// cont log-messages
      L     "SSA_LOG_Value_Queue".Input.Para_0099;	// message counter
      L     1;
      +I;
      T     "SSA_LOG_Value_Queue".Input.Para_0099;	// message counter
// Transform Basic Time to Local Time 
//      CALL  "BT_LT"
//       BT     :="DB Prozesszeit".Arbeitsbereich.dt1
//       WS_DAT :="RegelDB"
//       RET_VAL:=MW218
//       LT     :="RegelDB".LocalTime
// put timestamp into message
      CALL  FC 49 (
           $1                       := 1010,
           $2                       := 18,
           $3                       := 1005,
           $4                       := 462,
           $5                       := 8,
           $6                       := P#M 210.0);
///
      CALL  "SSA_MH_LogEntry_ActValue" (
           DBNumber                 := 1005);
E060: NOP   0;
///     
// Ereignis 26  Kommt         
      A     #EREIGNISBIT_26;
      FP    #Ereignis_26.FP_Kommt;
      JCN   E061;
// header
      L     #MessageType;
      T     "SSA_LOG_Value_Queue".Input.Header.SecType;	// type
      L     #MessageFormat;
      T     "SSA_LOG_Value_Queue".Input.Header.Format;	// format
      L     #JobNumber;
      T     "SSA_LOG_Value_Queue".Input.Para_0005;
      L     #processMinute;
      T     "SSA_LOG_Value_Queue".Input.Para_0007;
      L     #StepNumber;
      T     "SSA_LOG_Value_Queue".Input.Para_0008;
      L     #StepTimeMin;
      T     "SSA_LOG_Value_Queue".Input.Para_0009;
// values integer
      L     #EventObject_26;	// event-Nr
      T     "SSA_LOG_Value_Queue".Input.Para_0010;
      L     1;	// object-state coming
      T     "SSA_LOG_Value_Queue".Input.Para_0011;
      L     0;	// number additional param
      T     "SSA_LOG_Value_Queue".Input.Para_0012;
// cont log-messages
      L     "SSA_LOG_Value_Queue".Input.Para_0099;	// message counter
      L     1;
      +I;
      T     "SSA_LOG_Value_Queue".Input.Para_0099;	// message counter
// Transform Basic Time to Local Time 
//      CALL  "BT_LT"
//       BT     :="DB Prozesszeit".Arbeitsbereich.dt1
//       WS_DAT :="RegelDB"
//       RET_VAL:=MW218
//       LT     :="RegelDB".LocalTime
// put timestamp into message
      CALL  FC 49 (
           $1                       := 1010,
           $2                       := 18,
           $3                       := 1005,
           $4                       := 462,
           $5                       := 8,
           $6                       := P#M 210.0);
///
      CALL  "SSA_MH_LogEntry_ActValue" (
           DBNumber                 := 1005);
E061: NOP   0;
///
// Ereignis 26  Geht        
      A     #EREIGNISBIT_26;
      FN    #Ereignis_26.FN_Geht;
      JCN   E062;
// header
      L     #MessageType;
      T     "SSA_LOG_Value_Queue".Input.Header.SecType;	// type
      L     #MessageFormat;
      T     "SSA_LOG_Value_Queue".Input.Header.Format;	// format
      L     #JobNumber;
      T     "SSA_LOG_Value_Queue".Input.Para_0005;
      L     #processMinute;
      T     "SSA_LOG_Value_Queue".Input.Para_0007;
      L     #StepNumber;
      T     "SSA_LOG_Value_Queue".Input.Para_0008;
      L     #StepTimeMin;
      T     "SSA_LOG_Value_Queue".Input.Para_0009;
// values integer
      L     #EventObject_26;	// event-Nr
      T     "SSA_LOG_Value_Queue".Input.Para_0010;
      L     2;	// object-state going
      T     "SSA_LOG_Value_Queue".Input.Para_0011;
      L     0;	// number additional param
      T     "SSA_LOG_Value_Queue".Input.Para_0012;
// cont log-messages
      L     "SSA_LOG_Value_Queue".Input.Para_0099;	// message counter
      L     1;
      +I;
      T     "SSA_LOG_Value_Queue".Input.Para_0099;	// message counter
// Transform Basic Time to Local Time 
//      CALL  "BT_LT"
//       BT     :="DB Prozesszeit".Arbeitsbereich.dt1
//       WS_DAT :="RegelDB"
//       RET_VAL:=MW218
//       LT     :="RegelDB".LocalTime
// put timestamp into message
      CALL  FC 49 (
           $1                       := 1010,
           $2                       := 18,
           $3                       := 1005,
           $4                       := 462,
           $5                       := 8,
           $6                       := P#M 210.0);
///
      CALL  "SSA_MH_LogEntry_ActValue" (
           DBNumber                 := 1005);
E062: NOP   0;
///     
// Ereignis 27  Kommt         
      A     #EREIGNISBIT_27;
      FP    #Ereignis_27.FP_Kommt;
      JCN   E063;
/// header
      L     #MessageType;
      T     "SSA_LOG_Value_Queue".Input.Header.SecType;	// type
      L     #MessageFormat;
      T     "SSA_LOG_Value_Queue".Input.Header.Format;	// format
      L     #JobNumber;
      T     "SSA_LOG_Value_Queue".Input.Para_0005;
      L     #processMinute;
      T     "SSA_LOG_Value_Queue".Input.Para_0007;
      L     #StepNumber;
      T     "SSA_LOG_Value_Queue".Input.Para_0008;
      L     #StepTimeMin;
      T     "SSA_LOG_Value_Queue".Input.Para_0009;
// values integer
      L     #EventObject_27;	// event-Nr
      T     "SSA_LOG_Value_Queue".Input.Para_0010;
      L     1;	// object-state coming
      T     "SSA_LOG_Value_Queue".Input.Para_0011;
      L     0;	// number additional param
      T     "SSA_LOG_Value_Queue".Input.Para_0012;
// cont log-messages
      L     "SSA_LOG_Value_Queue".Input.Para_0099;	// message counter
      L     1;
      +I;
      T     "SSA_LOG_Value_Queue".Input.Para_0099;	// message counter
// Transform Basic Time to Local Time 
//      CALL  "BT_LT"
//       BT     :="DB Prozesszeit".Arbeitsbereich.dt1
//       WS_DAT :="RegelDB"
//       RET_VAL:=MW218
//       LT     :="RegelDB".LocalTime
// put timestamp into message
      CALL  FC 49 (
           $1                       := 1010,
           $2                       := 18,
           $3                       := 1005,
           $4                       := 462,
           $5                       := 8,
           $6                       := P#M 210.0);
///
      CALL  "SSA_MH_LogEntry_ActValue" (
           DBNumber                 := 1005);
E063: NOP   0;
///
// Ereignis 27  Geht        
      A     #EREIGNISBIT_27;
      FN    #Ereignis_27.FN_Geht;
      JCN   E064;
// header
      L     #MessageType;
      T     "SSA_LOG_Value_Queue".Input.Header.SecType;	// type
      L     #MessageFormat;
      T     "SSA_LOG_Value_Queue".Input.Header.Format;	// format
      L     #JobNumber;
      T     "SSA_LOG_Value_Queue".Input.Para_0005;
      L     #processMinute;
      T     "SSA_LOG_Value_Queue".Input.Para_0007;
      L     #StepNumber;
      T     "SSA_LOG_Value_Queue".Input.Para_0008;
      L     #StepTimeMin;
      T     "SSA_LOG_Value_Queue".Input.Para_0009;
// values integer
      L     #EventObject_27;	// event-Nr
      T     "SSA_LOG_Value_Queue".Input.Para_0010;
      L     2;	// object-state going
      T     "SSA_LOG_Value_Queue".Input.Para_0011;
      L     0;	// number additional param
      T     "SSA_LOG_Value_Queue".Input.Para_0012;
// cont log-messages
      L     "SSA_LOG_Value_Queue".Input.Para_0099;	// message counter
      L     1;
      +I;
      T     "SSA_LOG_Value_Queue".Input.Para_0099;	// message counter
// Transform Basic Time to Local Time 
//      CALL  "BT_LT"
//       BT     :="DB Prozesszeit".Arbeitsbereich.dt1
//       WS_DAT :="RegelDB"
//       RET_VAL:=MW218
//       LT     :="RegelDB".LocalTime
// put timestamp into message
      CALL  FC 49 (
           $1                       := 1010,
           $2                       := 18,
           $3                       := 1005,
           $4                       := 462,
           $5                       := 8,
           $6                       := P#M 210.0);
///
      CALL  "SSA_MH_LogEntry_ActValue" (
           DBNumber                 := 1005);
E064: NOP   0;
///     
// Ereignis 28  Kommt         
      A     #EREIGNISBIT_28;
      FP    #Ereignis_28.FP_Kommt;
      JCN   E065;
// header
      L     #MessageType;
      T     "SSA_LOG_Value_Queue".Input.Header.SecType;	// type
      L     #MessageFormat;
      T     "SSA_LOG_Value_Queue".Input.Header.Format;	// format
      L     #JobNumber;
      T     "SSA_LOG_Value_Queue".Input.Para_0005;
      L     #processMinute;
      T     "SSA_LOG_Value_Queue".Input.Para_0007;
      L     #StepNumber;
      T     "SSA_LOG_Value_Queue".Input.Para_0008;
      L     #StepTimeMin;
      T     "SSA_LOG_Value_Queue".Input.Para_0009;
// values integer
      L     #EventObject_28;	// event-Nr
      T     "SSA_LOG_Value_Queue".Input.Para_0010;
      L     1;	// object-state coming
      T     "SSA_LOG_Value_Queue".Input.Para_0011;
      L     0;	// number additional param
      T     "SSA_LOG_Value_Queue".Input.Para_0012;
// cont log-messages
      L     "SSA_LOG_Value_Queue".Input.Para_0099;	// message counter
      L     1;
      +I;
      T     "SSA_LOG_Value_Queue".Input.Para_0099;	// message counter
// Transform Basic Time to Local Time 
//      CALL  "BT_LT"
//       BT     :="DB Prozesszeit".Arbeitsbereich.dt1
//       WS_DAT :="RegelDB"
//       RET_VAL:=MW218
//       LT     :="RegelDB".LocalTime
// put timestamp into message
      CALL  FC 49 (
           $1                       := 1010,
           $2                       := 18,
           $3                       := 1005,
           $4                       := 462,
           $5                       := 8,
           $6                       := P#M 210.0);
///
      CALL  "SSA_MH_LogEntry_ActValue" (
           DBNumber                 := 1005);
E065: NOP   0;
///
// Ereignis 28  Geht        
      A     #EREIGNISBIT_28;
      FN    #Ereignis_28.FN_Geht;
      JCN   E066;
// header
      L     #MessageType;
      T     "SSA_LOG_Value_Queue".Input.Header.SecType;	// type
      L     #MessageFormat;
      T     "SSA_LOG_Value_Queue".Input.Header.Format;	// format
      L     #JobNumber;
      T     "SSA_LOG_Value_Queue".Input.Para_0005;
      L     #processMinute;
      T     "SSA_LOG_Value_Queue".Input.Para_0007;
      L     #StepNumber;
      T     "SSA_LOG_Value_Queue".Input.Para_0008;
      L     #StepTimeMin;
      T     "SSA_LOG_Value_Queue".Input.Para_0009;
// values integer
      L     #EventObject_28;	// event-Nr
      T     "SSA_LOG_Value_Queue".Input.Para_0010;
      L     2;	// object-state going
      T     "SSA_LOG_Value_Queue".Input.Para_0011;
      L     0;	// number additional param
      T     "SSA_LOG_Value_Queue".Input.Para_0012;
// cont log-messages
      L     "SSA_LOG_Value_Queue".Input.Para_0099;	// message counter
      L     1;
      +I;
      T     "SSA_LOG_Value_Queue".Input.Para_0099;	// message counter
// Transform Basic Time to Local Time 
//      CALL  "BT_LT"
//       BT     :="DB Prozesszeit".Arbeitsbereich.dt1
//       WS_DAT :="RegelDB"
//       RET_VAL:=MW218
//       LT     :="RegelDB".LocalTime
// put timestamp into message
      CALL  FC 49 (
           $1                       := 1010,
           $2                       := 18,
           $3                       := 1005,
           $4                       := 462,
           $5                       := 8,
           $6                       := P#M 210.0);
///
      CALL  "SSA_MH_LogEntry_ActValue" (
           DBNumber                 := 1005);
E066: NOP   0;
///     
// Ereignis 29  Kommt         
      A     #EREIGNISBIT_29;
      FP    #Ereignis_29.FP_Kommt;
      JCN   E067;
// header
      L     #MessageType;
      T     "SSA_LOG_Value_Queue".Input.Header.SecType;	// type
      L     #MessageFormat;
      T     "SSA_LOG_Value_Queue".Input.Header.Format;	// format
      L     #JobNumber;
      T     "SSA_LOG_Value_Queue".Input.Para_0005;
      L     #processMinute;
      T     "SSA_LOG_Value_Queue".Input.Para_0007;
      L     #StepNumber;
      T     "SSA_LOG_Value_Queue".Input.Para_0008;
      L     #StepTimeMin;
      T     "SSA_LOG_Value_Queue".Input.Para_0009;
// values integer
      L     #EventObject_29;	// event-Nr
      T     "SSA_LOG_Value_Queue".Input.Para_0010;
      L     1;	// object-state coming
      T     "SSA_LOG_Value_Queue".Input.Para_0011;
      L     0;	// number additional param
      T     "SSA_LOG_Value_Queue".Input.Para_0012;
// cont log-messages
      L     "SSA_LOG_Value_Queue".Input.Para_0099;	// message counter
      L     1;
      +I;
      T     "SSA_LOG_Value_Queue".Input.Para_0099;	// message counter
// Transform Basic Time to Local Time 
//      CALL  "BT_LT"
//       BT     :="DB Prozesszeit".Arbeitsbereich.dt1
//       WS_DAT :="RegelDB"
//       RET_VAL:=MW218
//       LT     :="RegelDB".LocalTime
// put timestamp into message
      CALL  FC 49 (
           $1                       := 1010,
           $2                       := 18,
           $3                       := 1005,
           $4                       := 462,
           $5                       := 8,
           $6                       := P#M 210.0);
///
      CALL  "SSA_MH_LogEntry_ActValue" (
           DBNumber                 := 1005);
E067: NOP   0;
///
// Ereignis 29  Geht        
      A     #EREIGNISBIT_29;
      FN    #Ereignis_29.FN_Geht;
      JCN   E068;
// header
      L     #MessageType;
      T     "SSA_LOG_Value_Queue".Input.Header.SecType;	// type
      L     #MessageFormat;
      T     "SSA_LOG_Value_Queue".Input.Header.Format;	// format
      L     #JobNumber;
      T     "SSA_LOG_Value_Queue".Input.Para_0005;
      L     #processMinute;
      T     "SSA_LOG_Value_Queue".Input.Para_0007;
      L     #StepNumber;
      T     "SSA_LOG_Value_Queue".Input.Para_0008;
      L     #StepTimeMin;
      T     "SSA_LOG_Value_Queue".Input.Para_0009;
// values integer
      L     #EventObject_29;	// event-Nr
      T     "SSA_LOG_Value_Queue".Input.Para_0010;
      L     2;	// object-state going
      T     "SSA_LOG_Value_Queue".Input.Para_0011;
      L     0;	// number additional param
      T     "SSA_LOG_Value_Queue".Input.Para_0012;
// cont log-messages
      L     "SSA_LOG_Value_Queue".Input.Para_0099;	// message counter
      L     1;
      +I;
      T     "SSA_LOG_Value_Queue".Input.Para_0099;	// message counter
// Transform Basic Time to Local Time 
//      CALL  "BT_LT"
//       BT     :="DB Prozesszeit".Arbeitsbereich.dt1
//       WS_DAT :="RegelDB"
//       RET_VAL:=MW218
//       LT     :="RegelDB".LocalTime
// put timestamp into message
      CALL  FC 49 (
           $1                       := 1010,
           $2                       := 18,
           $3                       := 1005,
           $4                       := 462,
           $5                       := 8,
           $6                       := P#M 210.0);
///
      CALL  "SSA_MH_LogEntry_ActValue" (
           DBNumber                 := 1005);
E068: NOP   0;
///     
// Ereignis 30  Kommt         
      A     #EREIGNISBIT_30;
      FP    #Ereignis_30.FP_Kommt;
      JCN   E069;
// header
      L     #MessageType;
      T     "SSA_LOG_Value_Queue".Input.Header.SecType;	// type
      L     #MessageFormat;
      T     "SSA_LOG_Value_Queue".Input.Header.Format;	// format
      L     #JobNumber;
      T     "SSA_LOG_Value_Queue".Input.Para_0005;
      L     #processMinute;
      T     "SSA_LOG_Value_Queue".Input.Para_0007;
      L     #StepNumber;
      T     "SSA_LOG_Value_Queue".Input.Para_0008;
      L     #StepTimeMin;
      T     "SSA_LOG_Value_Queue".Input.Para_0009;
// values integer
      L     #EventObject_30;	// event-Nr
      T     "SSA_LOG_Value_Queue".Input.Para_0010;
      L     1;	// object-state coming
      T     "SSA_LOG_Value_Queue".Input.Para_0011;
      L     0;	// number additional param
      T     "SSA_LOG_Value_Queue".Input.Para_0012;
// cont log-messages
      L     "SSA_LOG_Value_Queue".Input.Para_0099;	// message counter
      L     1;
      +I;
      T     "SSA_LOG_Value_Queue".Input.Para_0099;	// message counter
// Transform Basic Time to Local Time 
//      CALL  "BT_LT"
//       BT     :="DB Prozesszeit".Arbeitsbereich.dt1
//       WS_DAT :="RegelDB"
//       RET_VAL:=MW218
//       LT     :="RegelDB".LocalTime
// put timestamp into message
      CALL  FC 49 (
           $1                       := 1010,
           $2                       := 18,
           $3                       := 1005,
           $4                       := 462,
           $5                       := 8,
           $6                       := P#M 210.0);
///
      CALL  "SSA_MH_LogEntry_ActValue" (
           DBNumber                 := 1005);
E069: NOP   0;
///
// Ereignis 30  Geht        
      A     #EREIGNISBIT_30;
      FN    #Ereignis_30.FN_Geht;
      JCN   E070;
// header
      L     #MessageType;
      T     "SSA_LOG_Value_Queue".Input.Header.SecType;	// type
      L     #MessageFormat;
      T     "SSA_LOG_Value_Queue".Input.Header.Format;	// format
      L     #JobNumber;
      T     "SSA_LOG_Value_Queue".Input.Para_0005;
      L     #processMinute;
      T     "SSA_LOG_Value_Queue".Input.Para_0007;
      L     #StepNumber;
      T     "SSA_LOG_Value_Queue".Input.Para_0008;
      L     #StepTimeMin;
      T     "SSA_LOG_Value_Queue".Input.Para_0009;
// values integer
      L     #EventObject_30;	// event-Nr
      T     "SSA_LOG_Value_Queue".Input.Para_0010;
      L     2;	// object-state going
      T     "SSA_LOG_Value_Queue".Input.Para_0011;
      L     0;	// number additional param
      T     "SSA_LOG_Value_Queue".Input.Para_0012;
// cont log-messages
      L     "SSA_LOG_Value_Queue".Input.Para_0099;	// message counter
      L     1;
      +I;
      T     "SSA_LOG_Value_Queue".Input.Para_0099;	// message counter
// Transform Basic Time to Local Time 
//      CALL  "BT_LT"
//       BT     :="DB Prozesszeit".Arbeitsbereich.dt1
//       WS_DAT :="RegelDB"
//       RET_VAL:=MW218
//       LT     :="RegelDB".LocalTime
// put timestamp into message
      CALL  FC 49 (
           $1                       := 1010,
           $2                       := 18,
           $3                       := 1005,
           $4                       := 462,
           $5                       := 8,
           $6                       := P#M 210.0);
///
      CALL  "SSA_MH_LogEntry_ActValue" (
           DBNumber                 := 1005);
E070: NOP   0;
///     
NETWORK
TITLE = create events for batchprotokoll 
//event Nr. 121 - 130 are  events in job-protocol
///
// Ereignis 31  Kommt         
      A     #EREIGNISBIT_31;
      FP    #Ereignis_31.FP_Kommt;
      JCN   E071;
// header
      L     #MessageType;
      T     "SSA_LOG_Value_Queue".Input.Header.SecType;	// type
      L     #MessageFormat;
      T     "SSA_LOG_Value_Queue".Input.Header.Format;	// format
      L     #JobNumber;
      T     "SSA_LOG_Value_Queue".Input.Para_0005;
      L     #processMinute;
      T     "SSA_LOG_Value_Queue".Input.Para_0007;
      L     #StepNumber;
      T     "SSA_LOG_Value_Queue".Input.Para_0008;
      L     #StepTimeMin;
      T     "SSA_LOG_Value_Queue".Input.Para_0009;
// values integer
      L     #EventObject_31;	// event-Nr
      T     "SSA_LOG_Value_Queue".Input.Para_0010;
      L     1;	// object-state coming
      T     "SSA_LOG_Value_Queue".Input.Para_0011;
      L     0;	// number additional param
      T     "SSA_LOG_Value_Queue".Input.Para_0012;
// cont log-messages
      L     "SSA_LOG_Value_Queue".Input.Para_0099;	// message counter
      L     1;
      +I;
      T     "SSA_LOG_Value_Queue".Input.Para_0099;	// message counter
// Transform Basic Time to Local Time 
//      CALL  "BT_LT"
//       BT     :="DB Prozesszeit".Arbeitsbereich.dt1
//       WS_DAT :="RegelDB"
//       RET_VAL:=MW218
//       LT     :="RegelDB".LocalTime
// put timestamp into message
      CALL  FC 49 (
           $1                       := 1010,
           $2                       := 18,
           $3                       := 1005,
           $4                       := 462,
           $5                       := 8,
           $6                       := P#M 210.0);
///
      CALL  "SSA_MH_LogEntry_ActValue" (
           DBNumber                 := 1005);
E071: NOP   0;
///
// Ereignis 31  Geht        
      A     #EREIGNISBIT_31;
      FN    #Ereignis_31.FN_Geht;
      JCN   E072;
// header
      L     #MessageType;
      T     "SSA_LOG_Value_Queue".Input.Header.SecType;	// type
      L     #MessageFormat;
      T     "SSA_LOG_Value_Queue".Input.Header.Format;	// format
      L     #JobNumber;
      T     "SSA_LOG_Value_Queue".Input.Para_0005;
      L     #processMinute;
      T     "SSA_LOG_Value_Queue".Input.Para_0007;
      L     #StepNumber;
      T     "SSA_LOG_Value_Queue".Input.Para_0008;
      L     #StepTimeMin;
      T     "SSA_LOG_Value_Queue".Input.Para_0009;
// values integer
      L     #EventObject_31;	// event-Nr
      T     "SSA_LOG_Value_Queue".Input.Para_0010;
      L     2;	// object-state going
      T     "SSA_LOG_Value_Queue".Input.Para_0011;
      L     0;	// number additional param
      T     "SSA_LOG_Value_Queue".Input.Para_0012;
// cont log-messages
      L     "SSA_LOG_Value_Queue".Input.Para_0099;	// message counter
      L     1;
      +I;
      T     "SSA_LOG_Value_Queue".Input.Para_0099;	// message counter
// Transform Basic Time to Local Time 
//      CALL  "BT_LT"
//       BT     :="DB Prozesszeit".Arbeitsbereich.dt1
//       WS_DAT :="RegelDB"
//       RET_VAL:=MW218
//       LT     :="RegelDB".LocalTime
// put timestamp into message
      CALL  FC 49 (
           $1                       := 1010,
           $2                       := 18,
           $3                       := 1005,
           $4                       := 462,
           $5                       := 8,
           $6                       := P#M 210.0);
///
      CALL  "SSA_MH_LogEntry_ActValue" (
           DBNumber                 := 1005);
E072: NOP   0;
///     
// Ereignis 32  Kommt         
      A     #EREIGNISBIT_32;
      FP    #Ereignis_32.FP_Kommt;
      JCN   E073;
// header
      L     #MessageType;
      T     "SSA_LOG_Value_Queue".Input.Header.SecType;	// type
      L     #MessageFormat;
      T     "SSA_LOG_Value_Queue".Input.Header.Format;	// format
      L     #JobNumber;
      T     "SSA_LOG_Value_Queue".Input.Para_0005;
      L     #processMinute;
      T     "SSA_LOG_Value_Queue".Input.Para_0007;
      L     #StepNumber;
      T     "SSA_LOG_Value_Queue".Input.Para_0008;
      L     #StepTimeMin;
      T     "SSA_LOG_Value_Queue".Input.Para_0009;
// values integer
      L     #EventObject_32;	// event-Nr
      T     "SSA_LOG_Value_Queue".Input.Para_0010;
      L     1;	// object-state coming
      T     "SSA_LOG_Value_Queue".Input.Para_0011;
      L     0;	// number additional param
      T     "SSA_LOG_Value_Queue".Input.Para_0012;
// cont log-messages
      L     "SSA_LOG_Value_Queue".Input.Para_0099;	// message counter
      L     1;
      +I;
      T     "SSA_LOG_Value_Queue".Input.Para_0099;	// message counter
// Transform Basic Time to Local Time 
//      CALL  "BT_LT"
//       BT     :="DB Prozesszeit".Arbeitsbereich.dt1
//       WS_DAT :="RegelDB"
//       RET_VAL:=MW218
//       LT     :="RegelDB".LocalTime
// put timestamp into message
      CALL  FC 49 (
           $1                       := 1010,
           $2                       := 18,
           $3                       := 1005,
           $4                       := 462,
           $5                       := 8,
           $6                       := P#M 210.0);
///
      CALL  "SSA_MH_LogEntry_ActValue" (
           DBNumber                 := 1005);
E073: NOP   0;
///
// Ereignis 32  Geht        
      A     #EREIGNISBIT_32;
      FN    #Ereignis_32.FN_Geht;
      JCN   E074;
// header
      L     #MessageType;
      T     "SSA_LOG_Value_Queue".Input.Header.SecType;	// type
      L     #MessageFormat;
      T     "SSA_LOG_Value_Queue".Input.Header.Format;	// format
      L     #JobNumber;
      T     "SSA_LOG_Value_Queue".Input.Para_0005;
      L     #processMinute;
      T     "SSA_LOG_Value_Queue".Input.Para_0007;
      L     #StepNumber;
      T     "SSA_LOG_Value_Queue".Input.Para_0008;
      L     #StepTimeMin;
      T     "SSA_LOG_Value_Queue".Input.Para_0009;
// values integer
      L     #EventObject_32;	// event-Nr
      T     "SSA_LOG_Value_Queue".Input.Para_0010;
      L     2;	// object-state going
      T     "SSA_LOG_Value_Queue".Input.Para_0011;
      L     0;	// number additional param
      T     "SSA_LOG_Value_Queue".Input.Para_0012;
// cont log-messages
      L     "SSA_LOG_Value_Queue".Input.Para_0099;	// message counter
      L     1;
      +I;
      T     "SSA_LOG_Value_Queue".Input.Para_0099;	// message counter
// Transform Basic Time to Local Time 
//      CALL  "BT_LT"
//       BT     :="DB Prozesszeit".Arbeitsbereich.dt1
//       WS_DAT :="RegelDB"
//       RET_VAL:=MW218
//       LT     :="RegelDB".LocalTime
// put timestamp into message
      CALL  FC 49 (
           $1                       := 1010,
           $2                       := 18,
           $3                       := 1005,
           $4                       := 462,
           $5                       := 8,
           $6                       := P#M 210.0);
///
      CALL  "SSA_MH_LogEntry_ActValue" (
           DBNumber                 := 1005);
E074: NOP   0;
///     
// Ereignis 33  Kommt         
      A     #EREIGNISBIT_33;
      FP    #Ereignis_33.FP_Kommt;
      JCN   E075;
// header
      L     #MessageType;
      T     "SSA_LOG_Value_Queue".Input.Header.SecType;	// type
      L     #MessageFormat;
      T     "SSA_LOG_Value_Queue".Input.Header.Format;	// format
      L     #JobNumber;
      T     "SSA_LOG_Value_Queue".Input.Para_0005;
      L     #processMinute;
      T     "SSA_LOG_Value_Queue".Input.Para_0007;
      L     #StepNumber;
      T     "SSA_LOG_Value_Queue".Input.Para_0008;
      L     #StepTimeMin;
      T     "SSA_LOG_Value_Queue".Input.Para_0009;
// values integer
      L     #EventObject_33;	// event-Nr
      T     "SSA_LOG_Value_Queue".Input.Para_0010;
      L     1;	// object-state coming
      T     "SSA_LOG_Value_Queue".Input.Para_0011;
      L     0;	// number additional param
      T     "SSA_LOG_Value_Queue".Input.Para_0012;
// cont log-messages
      L     "SSA_LOG_Value_Queue".Input.Para_0099;	// message counter
      L     1;
      +I;
      T     "SSA_LOG_Value_Queue".Input.Para_0099;	// message counter
// Transform Basic Time to Local Time 
//      CALL  "BT_LT"
//       BT     :="DB Prozesszeit".Arbeitsbereich.dt1
//       WS_DAT :="RegelDB"
//       RET_VAL:=MW218
//       LT     :="RegelDB".LocalTime
// put timestamp into message
      CALL  FC 49 (
           $1                       := 1010,
           $2                       := 18,
           $3                       := 1005,
           $4                       := 462,
           $5                       := 8,
           $6                       := P#M 210.0);
///
      CALL  "SSA_MH_LogEntry_ActValue" (
           DBNumber                 := 1005);
E075: NOP   0;
///
// Ereignis 33  Geht        
      A     #EREIGNISBIT_33;
      FN    #Ereignis_33.FN_Geht;
      JCN   E076;
// header
      L     #MessageType;
      T     "SSA_LOG_Value_Queue".Input.Header.SecType;	// type
      L     #MessageFormat;
      T     "SSA_LOG_Value_Queue".Input.Header.Format;	// format
      L     #JobNumber;
      T     "SSA_LOG_Value_Queue".Input.Para_0005;
      L     #processMinute;
      T     "SSA_LOG_Value_Queue".Input.Para_0007;
      L     #StepNumber;
      T     "SSA_LOG_Value_Queue".Input.Para_0008;
      L     #StepTimeMin;
      T     "SSA_LOG_Value_Queue".Input.Para_0009;
// values integer
      L     #EventObject_33;	// event-Nr
      T     "SSA_LOG_Value_Queue".Input.Para_0010;
      L     2;	// object-state going
      T     "SSA_LOG_Value_Queue".Input.Para_0011;
      L     0;	// number additional param
      T     "SSA_LOG_Value_Queue".Input.Para_0012;
// cont log-messages
      L     "SSA_LOG_Value_Queue".Input.Para_0099;	// message counter
      L     1;
      +I;
      T     "SSA_LOG_Value_Queue".Input.Para_0099;	// message counter
// Transform Basic Time to Local Time 
//      CALL  "BT_LT"
//       BT     :="DB Prozesszeit".Arbeitsbereich.dt1
//       WS_DAT :="RegelDB"
//       RET_VAL:=MW218
//       LT     :="RegelDB".LocalTime
// put timestamp into message
      CALL  FC 49 (
           $1                       := 1010,
           $2                       := 18,
           $3                       := 1005,
           $4                       := 462,
           $5                       := 8,
           $6                       := P#M 210.0);
///
      CALL  "SSA_MH_LogEntry_ActValue" (
           DBNumber                 := 1005);
E076: NOP   0;
///     
// Ereignis 34  Kommt         
      A     #EREIGNISBIT_34;
      FP    #Ereignis_34.FP_Kommt;
      JCN   E077;
// header
      L     #MessageType;
      T     "SSA_LOG_Value_Queue".Input.Header.SecType;	// type
      L     #MessageFormat;
      T     "SSA_LOG_Value_Queue".Input.Header.Format;	// format
      L     #JobNumber;
      T     "SSA_LOG_Value_Queue".Input.Para_0005;
      L     #processMinute;
      T     "SSA_LOG_Value_Queue".Input.Para_0007;
      L     #StepNumber;
      T     "SSA_LOG_Value_Queue".Input.Para_0008;
      L     #StepTimeMin;
      T     "SSA_LOG_Value_Queue".Input.Para_0009;
// values integer
      L     #EventObject_34;	// event-Nr
      T     "SSA_LOG_Value_Queue".Input.Para_0010;
      L     1;	// object-state coming
      T     "SSA_LOG_Value_Queue".Input.Para_0011;
      L     0;	// number additional param
      T     "SSA_LOG_Value_Queue".Input.Para_0012;
// cont log-messages
      L     "SSA_LOG_Value_Queue".Input.Para_0099;	// message counter
      L     1;
      +I;
      T     "SSA_LOG_Value_Queue".Input.Para_0099;	// message counter
// Transform Basic Time to Local Time 
//      CALL  "BT_LT"
//       BT     :="DB Prozesszeit".Arbeitsbereich.dt1
//       WS_DAT :="RegelDB"
//       RET_VAL:=MW218
//       LT     :="RegelDB".LocalTime
// put timestamp into message
      CALL  FC 49 (
           $1                       := 1010,
           $2                       := 18,
           $3                       := 1005,
           $4                       := 462,
           $5                       := 8,
           $6                       := P#M 210.0);
///
      CALL  "SSA_MH_LogEntry_ActValue" (
           DBNumber                 := 1005);
E077: NOP   0;
///
// Ereignis 34  Geht        
      A     #EREIGNISBIT_34;
      FN    #Ereignis_34.FN_Geht;
      JCN   E078;
// header
      L     #MessageType;
      T     "SSA_LOG_Value_Queue".Input.Header.SecType;	// type
      L     #MessageFormat;
      T     "SSA_LOG_Value_Queue".Input.Header.Format;	// format
      L     #JobNumber;
      T     "SSA_LOG_Value_Queue".Input.Para_0005;
      L     #processMinute;
      T     "SSA_LOG_Value_Queue".Input.Para_0007;
      L     #StepNumber;
      T     "SSA_LOG_Value_Queue".Input.Para_0008;
      L     #StepTimeMin;
      T     "SSA_LOG_Value_Queue".Input.Para_0009;
// values integer
      L     #EventObject_34;	// event-Nr
      T     "SSA_LOG_Value_Queue".Input.Para_0010;
      L     2;	// object-state going
      T     "SSA_LOG_Value_Queue".Input.Para_0011;
      L     0;	// number additional param
      T     "SSA_LOG_Value_Queue".Input.Para_0012;
// cont log-messages
      L     "SSA_LOG_Value_Queue".Input.Para_0099;	// message counter
      L     1;
      +I;
      T     "SSA_LOG_Value_Queue".Input.Para_0099;	// message counter
// Transform Basic Time to Local Time 
//      CALL  "BT_LT"
//       BT     :="DB Prozesszeit".Arbeitsbereich.dt1
//       WS_DAT :="RegelDB"
//       RET_VAL:=MW218
//       LT     :="RegelDB".LocalTime
// put timestamp into message
      CALL  FC 49 (
           $1                       := 1010,
           $2                       := 18,
           $3                       := 1005,
           $4                       := 462,
           $5                       := 8,
           $6                       := P#M 210.0);
///
      CALL  "SSA_MH_LogEntry_ActValue" (
           DBNumber                 := 1005);
E078: NOP   0;
///     
// Ereignis 35  Kommt         
      A     #EREIGNISBIT_35;
      FP    #Ereignis_35.FP_Kommt;
      JCN   E079;
// header
      L     #MessageType;
      T     "SSA_LOG_Value_Queue".Input.Header.SecType;	// type
      L     #MessageFormat;
      T     "SSA_LOG_Value_Queue".Input.Header.Format;	// format
      L     #JobNumber;
      T     "SSA_LOG_Value_Queue".Input.Para_0005;
      L     #processMinute;
      T     "SSA_LOG_Value_Queue".Input.Para_0007;
      L     #StepNumber;
      T     "SSA_LOG_Value_Queue".Input.Para_0008;
      L     #StepTimeMin;
      T     "SSA_LOG_Value_Queue".Input.Para_0009;
// values integer
      L     #EventObject_35;	// event-Nr
      T     "SSA_LOG_Value_Queue".Input.Para_0010;
      L     1;	// object-state coming
      T     "SSA_LOG_Value_Queue".Input.Para_0011;
      L     0;	// number additional param
      T     "SSA_LOG_Value_Queue".Input.Para_0012;
// cont log-messages
      L     "SSA_LOG_Value_Queue".Input.Para_0099;	// message counter
      L     1;
      +I;
      T     "SSA_LOG_Value_Queue".Input.Para_0099;	// message counter
// Transform Basic Time to Local Time 
//      CALL  "BT_LT"
//       BT     :="DB Prozesszeit".Arbeitsbereich.dt1
//       WS_DAT :="RegelDB"
//       RET_VAL:=MW218
//       LT     :="RegelDB".LocalTime
// put timestamp into message
      CALL  FC 49 (
           $1                       := 1010,
           $2                       := 18,
           $3                       := 1005,
           $4                       := 462,
           $5                       := 8,
           $6                       := P#M 210.0);
///
      CALL  "SSA_MH_LogEntry_ActValue" (
           DBNumber                 := 1005);
E079: NOP   0;
///
// Ereignis 35  Geht        
      A     #EREIGNISBIT_35;
      FN    #Ereignis_35.FN_Geht;
      JCN   E080;
// header
      L     #MessageType;
      T     "SSA_LOG_Value_Queue".Input.Header.SecType;	// type
      L     #MessageFormat;
      T     "SSA_LOG_Value_Queue".Input.Header.Format;	// format
      L     #JobNumber;
      T     "SSA_LOG_Value_Queue".Input.Para_0005;
      L     #processMinute;
      T     "SSA_LOG_Value_Queue".Input.Para_0007;
      L     #StepNumber;
      T     "SSA_LOG_Value_Queue".Input.Para_0008;
      L     #StepTimeMin;
      T     "SSA_LOG_Value_Queue".Input.Para_0009;
// values integer
      L     #EventObject_35;	// event-Nr
      T     "SSA_LOG_Value_Queue".Input.Para_0010;
      L     2;	// object-state going
      T     "SSA_LOG_Value_Queue".Input.Para_0011;
      L     0;	// number additional param
      T     "SSA_LOG_Value_Queue".Input.Para_0012;
// cont log-messages
      L     "SSA_LOG_Value_Queue".Input.Para_0099;	// message counter
      L     1;
      +I;
      T     "SSA_LOG_Value_Queue".Input.Para_0099;	// message counter
// Transform Basic Time to Local Time 
//      CALL  "BT_LT"
//       BT     :="DB Prozesszeit".Arbeitsbereich.dt1
//       WS_DAT :="RegelDB"
//       RET_VAL:=MW218
//       LT     :="RegelDB".LocalTime
// put timestamp into message
      CALL  FC 49 (
           $1                       := 1010,
           $2                       := 18,
           $3                       := 1005,
           $4                       := 462,
           $5                       := 8,
           $6                       := P#M 210.0);
///
      CALL  "SSA_MH_LogEntry_ActValue" (
           DBNumber                 := 1005);
E080: NOP   0;
///     
// Ereignis 36  Kommt         
      A     #EREIGNISBIT_36;
      FP    #Ereignis_36.FP_Kommt;
      JCN   E081;
// header
      L     #MessageType;
      T     "SSA_LOG_Value_Queue".Input.Header.SecType;	// type
      L     #MessageFormat;
      T     "SSA_LOG_Value_Queue".Input.Header.Format;	// format
      L     #JobNumber;
      T     "SSA_LOG_Value_Queue".Input.Para_0005;
      L     #processMinute;
      T     "SSA_LOG_Value_Queue".Input.Para_0007;
      L     #StepNumber;
      T     "SSA_LOG_Value_Queue".Input.Para_0008;
      L     #StepTimeMin;
      T     "SSA_LOG_Value_Queue".Input.Para_0009;
// values integer
      L     #EventObject_36;	// event-Nr
      T     "SSA_LOG_Value_Queue".Input.Para_0010;
      L     1;	// object-state coming
      T     "SSA_LOG_Value_Queue".Input.Para_0011;
      L     0;	// number additional param
      T     "SSA_LOG_Value_Queue".Input.Para_0012;
// cont log-messages
      L     "SSA_LOG_Value_Queue".Input.Para_0099;	// message counter
      L     1;
      +I;
      T     "SSA_LOG_Value_Queue".Input.Para_0099;	// message counter
// Transform Basic Time to Local Time 
//      CALL  "BT_LT"
//       BT     :="DB Prozesszeit".Arbeitsbereich.dt1
//       WS_DAT :="RegelDB"
//       RET_VAL:=MW218
//       LT     :="RegelDB".LocalTime
// put timestamp into message
      CALL  FC 49 (
           $1                       := 1010,
           $2                       := 18,
           $3                       := 1005,
           $4                       := 462,
           $5                       := 8,
           $6                       := P#M 210.0);
///
      CALL  "SSA_MH_LogEntry_ActValue" (
           DBNumber                 := 1005);
E081: NOP   0;
///
// Ereignis 36  Geht        
      A     #EREIGNISBIT_36;
      FN    #Ereignis_36.FN_Geht;
      JCN   E082;
// header
      L     #MessageType;
      T     "SSA_LOG_Value_Queue".Input.Header.SecType;	// type
      L     #MessageFormat;
      T     "SSA_LOG_Value_Queue".Input.Header.Format;	// format
      L     #JobNumber;
      T     "SSA_LOG_Value_Queue".Input.Para_0005;
      L     #processMinute;
      T     "SSA_LOG_Value_Queue".Input.Para_0007;
      L     #StepNumber;
      T     "SSA_LOG_Value_Queue".Input.Para_0008;
      L     #StepTimeMin;
      T     "SSA_LOG_Value_Queue".Input.Para_0009;
// values integer
      L     #EventObject_36;	// event-Nr
      T     "SSA_LOG_Value_Queue".Input.Para_0010;
      L     2;	// object-state going
      T     "SSA_LOG_Value_Queue".Input.Para_0011;
      L     0;	// number additional param
      T     "SSA_LOG_Value_Queue".Input.Para_0012;
// cont log-messages
      L     "SSA_LOG_Value_Queue".Input.Para_0099;	// message counter
      L     1;
      +I;
      T     "SSA_LOG_Value_Queue".Input.Para_0099;	// message counter
// Transform Basic Time to Local Time 
//      CALL  "BT_LT"
//       BT     :="DB Prozesszeit".Arbeitsbereich.dt1
//       WS_DAT :="RegelDB"
//       RET_VAL:=MW218
//       LT     :="RegelDB".LocalTime
// put timestamp into message
      CALL  FC 49 (
           $1                       := 1010,
           $2                       := 18,
           $3                       := 1005,
           $4                       := 462,
           $5                       := 8,
           $6                       := P#M 210.0);
///
      CALL  "SSA_MH_LogEntry_ActValue" (
           DBNumber                 := 1005);
E082: NOP   0;
///     
// Ereignis 37  Kommt         
      A     #EREIGNISBIT_37;
      FP    #Ereignis_37.FP_Kommt;
      JCN   E083;
// header
      L     #MessageType;
      T     "SSA_LOG_Value_Queue".Input.Header.SecType;	// type
      L     #MessageFormat;
      T     "SSA_LOG_Value_Queue".Input.Header.Format;	// format
      L     #JobNumber;
      T     "SSA_LOG_Value_Queue".Input.Para_0005;
      L     #processMinute;
      T     "SSA_LOG_Value_Queue".Input.Para_0007;
      L     #StepNumber;
      T     "SSA_LOG_Value_Queue".Input.Para_0008;
      L     #StepTimeMin;
      T     "SSA_LOG_Value_Queue".Input.Para_0009;
// values integer
      L     #EventObject_37;	// event-Nr
      T     "SSA_LOG_Value_Queue".Input.Para_0010;
      L     1;	// object-state coming
      T     "SSA_LOG_Value_Queue".Input.Para_0011;
      L     0;	// number additional param
      T     "SSA_LOG_Value_Queue".Input.Para_0012;
// cont log-messages
      L     "SSA_LOG_Value_Queue".Input.Para_0099;	// message counter
      L     1;
      +I;
      T     "SSA_LOG_Value_Queue".Input.Para_0099;	// message counter
// Transform Basic Time to Local Time 
//      CALL  "BT_LT"
//       BT     :="DB Prozesszeit".Arbeitsbereich.dt1
//       WS_DAT :="RegelDB"
//       RET_VAL:=MW218
//       LT     :="RegelDB".LocalTime
// put timestamp into message
      CALL  FC 49 (
           $1                       := 1010,
           $2                       := 18,
           $3                       := 1005,
           $4                       := 462,
           $5                       := 8,
           $6                       := P#M 210.0);
///
      CALL  "SSA_MH_LogEntry_ActValue" (
           DBNumber                 := 1005);
E083: NOP   0;
///
// Ereignis 37  Geht        
      A     #EREIGNISBIT_37;
      FN    #Ereignis_37.FN_Geht;
      JCN   E084;
// header
      L     #MessageType;
      T     "SSA_LOG_Value_Queue".Input.Header.SecType;	// type
      L     #MessageFormat;
      T     "SSA_LOG_Value_Queue".Input.Header.Format;	// format
      L     #JobNumber;
      T     "SSA_LOG_Value_Queue".Input.Para_0005;
      L     #processMinute;
      T     "SSA_LOG_Value_Queue".Input.Para_0007;
      L     #StepNumber;
      T     "SSA_LOG_Value_Queue".Input.Para_0008;
      L     #StepTimeMin;
      T     "SSA_LOG_Value_Queue".Input.Para_0009;
// values integer
      L     #EventObject_37;	// event-Nr
      T     "SSA_LOG_Value_Queue".Input.Para_0010;
      L     2;	// object-state going
      T     "SSA_LOG_Value_Queue".Input.Para_0011;
      L     0;	// number additional param
      T     "SSA_LOG_Value_Queue".Input.Para_0012;
// cont log-messages
      L     "SSA_LOG_Value_Queue".Input.Para_0099;	// message counter
      L     1;
      +I;
      T     "SSA_LOG_Value_Queue".Input.Para_0099;	// message counter
// Transform Basic Time to Local Time 
//      CALL  "BT_LT"
//       BT     :="DB Prozesszeit".Arbeitsbereich.dt1
//       WS_DAT :="RegelDB"
//       RET_VAL:=MW218
//       LT     :="RegelDB".LocalTime
// put timestamp into message
      CALL  FC 49 (
           $1                       := 1010,
           $2                       := 18,
           $3                       := 1005,
           $4                       := 462,
           $5                       := 8,
           $6                       := P#M 210.0);
///
      CALL  "SSA_MH_LogEntry_ActValue" (
           DBNumber                 := 1005);
E084: NOP   0;
///     
// Ereignis 38  Kommt         
      A     #EREIGNISBIT_38;
      FP    #Ereignis_38.FP_Kommt;
      JCN   E085;
// header
      L     #MessageType;
      T     "SSA_LOG_Value_Queue".Input.Header.SecType;	// type
      L     #MessageFormat;
      T     "SSA_LOG_Value_Queue".Input.Header.Format;	// format
      L     #JobNumber;
      T     "SSA_LOG_Value_Queue".Input.Para_0005;
      L     #processMinute;
      T     "SSA_LOG_Value_Queue".Input.Para_0007;
      L     #StepNumber;
      T     "SSA_LOG_Value_Queue".Input.Para_0008;
      L     #StepTimeMin;
      T     "SSA_LOG_Value_Queue".Input.Para_0009;
// values integer
      L     #EventObject_38;	// event-Nr
      T     "SSA_LOG_Value_Queue".Input.Para_0010;
      L     1;	// object-state coming
      T     "SSA_LOG_Value_Queue".Input.Para_0011;
      L     0;	// number additional param
      T     "SSA_LOG_Value_Queue".Input.Para_0012;
// cont log-messages
      L     "SSA_LOG_Value_Queue".Input.Para_0099;	// message counter
      L     1;
      +I;
      T     "SSA_LOG_Value_Queue".Input.Para_0099;	// message counter
// Transform Basic Time to Local Time 
//      CALL  "BT_LT"
//       BT     :="DB Prozesszeit".Arbeitsbereich.dt1
//       WS_DAT :="RegelDB"
//       RET_VAL:=MW218
//       LT     :="RegelDB".LocalTime
// put timestamp into message
      CALL  FC 49 (
           $1                       := 1010,
           $2                       := 18,
           $3                       := 1005,
           $4                       := 462,
           $5                       := 8,
           $6                       := P#M 210.0);
///
      CALL  "SSA_MH_LogEntry_ActValue" (
           DBNumber                 := 1005);
E085: NOP   0;
///
// Ereignis 38  Geht        
      A     #EREIGNISBIT_38;
      FN    #Ereignis_38.FN_Geht;
      JCN   E086;
// header
      L     #MessageType;
      T     "SSA_LOG_Value_Queue".Input.Header.SecType;	// type
      L     #MessageFormat;
      T     "SSA_LOG_Value_Queue".Input.Header.Format;	// format
      L     #JobNumber;
      T     "SSA_LOG_Value_Queue".Input.Para_0005;
      L     #processMinute;
      T     "SSA_LOG_Value_Queue".Input.Para_0007;
      L     #StepNumber;
      T     "SSA_LOG_Value_Queue".Input.Para_0008;
      L     #StepTimeMin;
      T     "SSA_LOG_Value_Queue".Input.Para_0009;
// values integer
      L     #EventObject_38;	// event-Nr
      T     "SSA_LOG_Value_Queue".Input.Para_0010;
      L     2;	// object-state going
      T     "SSA_LOG_Value_Queue".Input.Para_0011;
      L     0;	// number additional param
      T     "SSA_LOG_Value_Queue".Input.Para_0012;
// cont log-messages
      L     "SSA_LOG_Value_Queue".Input.Para_0099;	// message counter
      L     1;
      +I;
      T     "SSA_LOG_Value_Queue".Input.Para_0099;	// message counter
// Transform Basic Time to Local Time 
//      CALL  "BT_LT"
//       BT     :="DB Prozesszeit".Arbeitsbereich.dt1
//       WS_DAT :="RegelDB"
//       RET_VAL:=MW218
//       LT     :="RegelDB".LocalTime
// put timestamp into message
      CALL  FC 49 (
           $1                       := 1010,
           $2                       := 18,
           $3                       := 1005,
           $4                       := 462,
           $5                       := 8,
           $6                       := P#M 210.0);
///
      CALL  "SSA_MH_LogEntry_ActValue" (
           DBNumber                 := 1005);
E086: NOP   0;
///     
// Ereignis 39  Kommt         
      A     #EREIGNISBIT_39;
      FP    #Ereignis_39.FP_Kommt;
      JCN   E087;
// header
      L     #MessageType;
      T     "SSA_LOG_Value_Queue".Input.Header.SecType;	// type
      L     #MessageFormat;
      T     "SSA_LOG_Value_Queue".Input.Header.Format;	// format
      L     #JobNumber;
      T     "SSA_LOG_Value_Queue".Input.Para_0005;
      L     #processMinute;
      T     "SSA_LOG_Value_Queue".Input.Para_0007;
      L     #StepNumber;
      T     "SSA_LOG_Value_Queue".Input.Para_0008;
      L     #StepTimeMin;
      T     "SSA_LOG_Value_Queue".Input.Para_0009;
// values integer
      L     #EventObject_39;	// event-Nr
      T     "SSA_LOG_Value_Queue".Input.Para_0010;
      L     1;	// object-state coming
      T     "SSA_LOG_Value_Queue".Input.Para_0011;
      L     0;	// number additional param
      T     "SSA_LOG_Value_Queue".Input.Para_0012;
// cont log-messages
      L     "SSA_LOG_Value_Queue".Input.Para_0099;	// message counter
      L     1;
      +I;
      T     "SSA_LOG_Value_Queue".Input.Para_0099;	// message counter
// Transform Basic Time to Local Time 
//      CALL  "BT_LT"
//       BT     :="DB Prozesszeit".Arbeitsbereich.dt1
//       WS_DAT :="RegelDB"
//       RET_VAL:=MW218
//       LT     :="RegelDB".LocalTime
// put timestamp into message
      CALL  FC 49 (
           $1                       := 1010,
           $2                       := 18,
           $3                       := 1005,
           $4                       := 462,
           $5                       := 8,
           $6                       := P#M 210.0);
///
      CALL  "SSA_MH_LogEntry_ActValue" (
           DBNumber                 := 1005);
E087: NOP   0;
///
// Ereignis 39  Geht        
      A     #EREIGNISBIT_39;
      FN    #Ereignis_39.FN_Geht;
      JCN   E088;
// header
      L     #MessageType;
      T     "SSA_LOG_Value_Queue".Input.Header.SecType;	// type
      L     #MessageFormat;
      T     "SSA_LOG_Value_Queue".Input.Header.Format;	// format
      L     #JobNumber;
      T     "SSA_LOG_Value_Queue".Input.Para_0005;
      L     #processMinute;
      T     "SSA_LOG_Value_Queue".Input.Para_0007;
      L     #StepNumber;
      T     "SSA_LOG_Value_Queue".Input.Para_0008;
      L     #StepTimeMin;
      T     "SSA_LOG_Value_Queue".Input.Para_0009;
// values integer
      L     #EventObject_39;	// event-Nr
      T     "SSA_LOG_Value_Queue".Input.Para_0010;
      L     2;	// object-state going
      T     "SSA_LOG_Value_Queue".Input.Para_0011;
      L     0;	// number additional param
      T     "SSA_LOG_Value_Queue".Input.Para_0012;
// cont log-messages
      L     "SSA_LOG_Value_Queue".Input.Para_0099;	// message counter
      L     1;
      +I;
      T     "SSA_LOG_Value_Queue".Input.Para_0099;	// message counter
// Transform Basic Time to Local Time 
//      CALL  "BT_LT"
//       BT     :="DB Prozesszeit".Arbeitsbereich.dt1
//       WS_DAT :="RegelDB"
//       RET_VAL:=MW218
//       LT     :="RegelDB".LocalTime
// put timestamp into message
      CALL  FC 49 (
           $1                       := 1010,
           $2                       := 18,
           $3                       := 1005,
           $4                       := 462,
           $5                       := 8,
           $6                       := P#M 210.0);
///
      CALL  "SSA_MH_LogEntry_ActValue" (
           DBNumber                 := 1005);
E088: NOP   0;
///     
// Ereignis 40  Kommt         
      A     #EREIGNISBIT_40;
      FP    #Ereignis_40.FP_Kommt;
      JCN   E089;
// header
      L     #MessageType;
      T     "SSA_LOG_Value_Queue".Input.Header.SecType;	// type
      L     #MessageFormat;
      T     "SSA_LOG_Value_Queue".Input.Header.Format;	// format
      L     #JobNumber;
      T     "SSA_LOG_Value_Queue".Input.Para_0005;
      L     #processMinute;
      T     "SSA_LOG_Value_Queue".Input.Para_0007;
      L     #StepNumber;
      T     "SSA_LOG_Value_Queue".Input.Para_0008;
      L     #StepTimeMin;
      T     "SSA_LOG_Value_Queue".Input.Para_0009;
// values integer
      L     #EventObject_40;	// event-Nr
      T     "SSA_LOG_Value_Queue".Input.Para_0010;
      L     1;	// object-state coming
      T     "SSA_LOG_Value_Queue".Input.Para_0011;
      L     0;	// number additional param
      T     "SSA_LOG_Value_Queue".Input.Para_0012;
// cont log-messages
      L     "SSA_LOG_Value_Queue".Input.Para_0099;	// message counter
      L     1;
      +I;
      T     "SSA_LOG_Value_Queue".Input.Para_0099;	// message counter
// Transform Basic Time to Local Time 
//      CALL  "BT_LT"
//       BT     :="DB Prozesszeit".Arbeitsbereich.dt1
//       WS_DAT :="RegelDB"
//       RET_VAL:=MW218
//       LT     :="RegelDB".LocalTime
// put timestamp into message
      CALL  FC 49 (
           $1                       := 1010,
           $2                       := 18,
           $3                       := 1005,
           $4                       := 462,
           $5                       := 8,
           $6                       := P#M 210.0);
///
      CALL  "SSA_MH_LogEntry_ActValue" (
           DBNumber                 := 1005);
E089: NOP   0;
///
// Ereignis 40  Geht        
      A     #EREIGNISBIT_40;
      FN    #Ereignis_40.FN_Geht;
      JCN   E090;
// header
      L     #MessageType;
      T     "SSA_LOG_Value_Queue".Input.Header.SecType;	// type
      L     #MessageFormat;
      T     "SSA_LOG_Value_Queue".Input.Header.Format;	// format
      L     #JobNumber;
      T     "SSA_LOG_Value_Queue".Input.Para_0005;
      L     #processMinute;
      T     "SSA_LOG_Value_Queue".Input.Para_0007;
      L     #StepNumber;
      T     "SSA_LOG_Value_Queue".Input.Para_0008;
      L     #StepTimeMin;
      T     "SSA_LOG_Value_Queue".Input.Para_0009;
// values integer
      L     #EventObject_40;	// event-Nr
      T     "SSA_LOG_Value_Queue".Input.Para_0010;
      L     2;	// object-state going
      T     "SSA_LOG_Value_Queue".Input.Para_0011;
      L     0;	// number additional param
      T     "SSA_LOG_Value_Queue".Input.Para_0012;
// cont log-messages
      L     "SSA_LOG_Value_Queue".Input.Para_0099;	// message counter
      L     1;
      +I;
      T     "SSA_LOG_Value_Queue".Input.Para_0099;	// message counter
// Transform Basic Time to Local Time 
//      CALL  "BT_LT"
//       BT     :="DB Prozesszeit".Arbeitsbereich.dt1
//       WS_DAT :="RegelDB"
//       RET_VAL:=MW218
//       LT     :="RegelDB".LocalTime
// put timestamp into message
      CALL  FC 49 (
           $1                       := 1010,
           $2                       := 18,
           $3                       := 1005,
           $4                       := 462,
           $5                       := 8,
           $6                       := P#M 210.0);
///
      CALL  "SSA_MH_LogEntry_ActValue" (
           DBNumber                 := 1005);
E090: NOP   0;
///     
// Ereignis 41  Kommt         
      A     #EREIGNISBIT_41;
      FP    #Ereignis_41.FP_Kommt;
      JCN   E091;
// header
      L     #MessageType;
      T     "SSA_LOG_Value_Queue".Input.Header.SecType;	// type
      L     #MessageFormat;
      T     "SSA_LOG_Value_Queue".Input.Header.Format;	// format
      L     #JobNumber;
      T     "SSA_LOG_Value_Queue".Input.Para_0005;
      L     #processMinute;
      T     "SSA_LOG_Value_Queue".Input.Para_0007;
      L     #StepNumber;
      T     "SSA_LOG_Value_Queue".Input.Para_0008;
      L     #StepTimeMin;
      T     "SSA_LOG_Value_Queue".Input.Para_0009;
// values integer
      L     #EventObject_41;	// event-Nr
      T     "SSA_LOG_Value_Queue".Input.Para_0010;
      L     1;	// object-state coming
      T     "SSA_LOG_Value_Queue".Input.Para_0011;
      L     0;	// number additional param
      T     "SSA_LOG_Value_Queue".Input.Para_0012;
// cont log-messages
      L     "SSA_LOG_Value_Queue".Input.Para_0099;	// message counter
      L     1;
      +I;
      T     "SSA_LOG_Value_Queue".Input.Para_0099;	// message counter
// Transform Basic Time to Local Time 
//      CALL  "BT_LT"
//       BT     :="DB Prozesszeit".Arbeitsbereich.dt1
//       WS_DAT :="RegelDB"
//       RET_VAL:=MW218
//       LT     :="RegelDB".LocalTime
// put timestamp into message
      CALL  FC 49 (
           $1                       := 1010,
           $2                       := 18,
           $3                       := 1005,
           $4                       := 462,
           $5                       := 8,
           $6                       := P#M 210.0);
///
      CALL  "SSA_MH_LogEntry_ActValue" (
           DBNumber                 := 1005);
E091: NOP   0;
///
// Ereignis 41  Geht        
      A     #EREIGNISBIT_41;
      FN    #Ereignis_41.FN_Geht;
      JCN   E092;
// header
      L     #MessageType;
      T     "SSA_LOG_Value_Queue".Input.Header.SecType;	// type
      L     #MessageFormat;
      T     "SSA_LOG_Value_Queue".Input.Header.Format;	// format
      L     #JobNumber;
      T     "SSA_LOG_Value_Queue".Input.Para_0005;
      L     #processMinute;
      T     "SSA_LOG_Value_Queue".Input.Para_0007;
      L     #StepNumber;
      T     "SSA_LOG_Value_Queue".Input.Para_0008;
      L     #StepTimeMin;
      T     "SSA_LOG_Value_Queue".Input.Para_0009;
// values integer
      L     #EventObject_41;	// event-Nr
      T     "SSA_LOG_Value_Queue".Input.Para_0010;
      L     2;	// object-state going
      T     "SSA_LOG_Value_Queue".Input.Para_0011;
      L     0;	// number additional param
      T     "SSA_LOG_Value_Queue".Input.Para_0012;
// cont log-messages
      L     "SSA_LOG_Value_Queue".Input.Para_0099;	// message counter
      L     1;
      +I;
      T     "SSA_LOG_Value_Queue".Input.Para_0099;	// message counter
// Transform Basic Time to Local Time 
//      CALL  "BT_LT"
//       BT     :="DB Prozesszeit".Arbeitsbereich.dt1
//       WS_DAT :="RegelDB"
//       RET_VAL:=MW218
//       LT     :="RegelDB".LocalTime
// put timestamp into message
      CALL  FC 49 (
           $1                       := 1010,
           $2                       := 18,
           $3                       := 1005,
           $4                       := 462,
           $5                       := 8,
           $6                       := P#M 210.0);
///
      CALL  "SSA_MH_LogEntry_ActValue" (
           DBNumber                 := 1005);
E092: NOP   0;
///     
// Ereignis 42  Kommt         
      A     #EREIGNISBIT_42;
      FP    #Ereignis_42.FP_Kommt;
      JCN   E093;
// header
      L     #MessageType;
      T     "SSA_LOG_Value_Queue".Input.Header.SecType;	// type
      L     #MessageFormat;
      T     "SSA_LOG_Value_Queue".Input.Header.Format;	// format
      L     #JobNumber;
      T     "SSA_LOG_Value_Queue".Input.Para_0005;
      L     #processMinute;
      T     "SSA_LOG_Value_Queue".Input.Para_0007;
      L     #StepNumber;
      T     "SSA_LOG_Value_Queue".Input.Para_0008;
      L     #StepTimeMin;
      T     "SSA_LOG_Value_Queue".Input.Para_0009;
// values integer
      L     #EventObject_42;	// event-Nr
      T     "SSA_LOG_Value_Queue".Input.Para_0010;
      L     1;	// object-state coming
      T     "SSA_LOG_Value_Queue".Input.Para_0011;
      L     0;	// number additional param
      T     "SSA_LOG_Value_Queue".Input.Para_0012;
// cont log-messages
      L     "SSA_LOG_Value_Queue".Input.Para_0099;	// message counter
      L     1;
      +I;
      T     "SSA_LOG_Value_Queue".Input.Para_0099;	// message counter
// Transform Basic Time to Local Time 
//      CALL  "BT_LT"
//       BT     :="DB Prozesszeit".Arbeitsbereich.dt1
//       WS_DAT :="RegelDB"
//       RET_VAL:=MW218
//       LT     :="RegelDB".LocalTime
// put timestamp into message
      CALL  FC 49 (
           $1                       := 1010,
           $2                       := 18,
           $3                       := 1005,
           $4                       := 462,
           $5                       := 8,
           $6                       := P#M 210.0);
///
      CALL  "SSA_MH_LogEntry_ActValue" (
           DBNumber                 := 1005);
E093: NOP   0;
///
// Ereignis 42  Geht        
      A     #EREIGNISBIT_42;
      FN    #Ereignis_42.FN_Geht;
      JCN   E094;
// header
      L     #MessageType;
      T     "SSA_LOG_Value_Queue".Input.Header.SecType;	// type
      L     #MessageFormat;
      T     "SSA_LOG_Value_Queue".Input.Header.Format;	// format
      L     #JobNumber;
      T     "SSA_LOG_Value_Queue".Input.Para_0005;
      L     #processMinute;
      T     "SSA_LOG_Value_Queue".Input.Para_0007;
      L     #StepNumber;
      T     "SSA_LOG_Value_Queue".Input.Para_0008;
      L     #StepTimeMin;
      T     "SSA_LOG_Value_Queue".Input.Para_0009;
// values integer
      L     #EventObject_42;	// event-Nr
      T     "SSA_LOG_Value_Queue".Input.Para_0010;
      L     2;	// object-state going
      T     "SSA_LOG_Value_Queue".Input.Para_0011;
      L     0;	// number additional param
      T     "SSA_LOG_Value_Queue".Input.Para_0012;
// cont log-messages
      L     "SSA_LOG_Value_Queue".Input.Para_0099;	// message counter
      L     1;
      +I;
      T     "SSA_LOG_Value_Queue".Input.Para_0099;	// message counter
// Transform Basic Time to Local Time 
//      CALL  "BT_LT"
//       BT     :="DB Prozesszeit".Arbeitsbereich.dt1
//       WS_DAT :="RegelDB"
//       RET_VAL:=MW218
//       LT     :="RegelDB".LocalTime
// put timestamp into message
      CALL  FC 49 (
           $1                       := 1010,
           $2                       := 18,
           $3                       := 1005,
           $4                       := 462,
           $5                       := 8,
           $6                       := P#M 210.0);
///
      CALL  "SSA_MH_LogEntry_ActValue" (
           DBNumber                 := 1005);
E094: NOP   0;
///     
// Ereignis 43  Kommt         
      A     #EREIGNISBIT_43;
      FP    #Ereignis_43.FP_Kommt;
      JCN   E095;
// header
      L     #MessageType;
      T     "SSA_LOG_Value_Queue".Input.Header.SecType;	// type
      L     #MessageFormat;
      T     "SSA_LOG_Value_Queue".Input.Header.Format;	// format
      L     #JobNumber;
      T     "SSA_LOG_Value_Queue".Input.Para_0005;
      L     #processMinute;
      T     "SSA_LOG_Value_Queue".Input.Para_0007;
      L     #StepNumber;
      T     "SSA_LOG_Value_Queue".Input.Para_0008;
      L     #StepTimeMin;
      T     "SSA_LOG_Value_Queue".Input.Para_0009;
// values integer
      L     #EventObject_43;	// event-Nr
      T     "SSA_LOG_Value_Queue".Input.Para_0010;
      L     1;	// object-state coming
      T     "SSA_LOG_Value_Queue".Input.Para_0011;
      L     0;	// number additional param
      T     "SSA_LOG_Value_Queue".Input.Para_0012;
// cont log-messages
      L     "SSA_LOG_Value_Queue".Input.Para_0099;	// message counter
      L     1;
      +I;
      T     "SSA_LOG_Value_Queue".Input.Para_0099;	// message counter
// Transform Basic Time to Local Time 
//      CALL  "BT_LT"
//       BT     :="DB Prozesszeit".Arbeitsbereich.dt1
//       WS_DAT :="RegelDB"
//       RET_VAL:=MW218
//       LT     :="RegelDB".LocalTime
// put timestamp into message
      CALL  FC 49 (
           $1                       := 1010,
           $2                       := 18,
           $3                       := 1005,
           $4                       := 462,
           $5                       := 8,
           $6                       := P#M 210.0);
///
      CALL  "SSA_MH_LogEntry_ActValue" (
           DBNumber                 := 1005);
E095: NOP   0;
///
// Ereignis 43  Geht        
      A     #EREIGNISBIT_43;
      FN    #Ereignis_43.FN_Geht;
      JCN   E096;
// header
      L     #MessageType;
      T     "SSA_LOG_Value_Queue".Input.Header.SecType;	// type
      L     #MessageFormat;
      T     "SSA_LOG_Value_Queue".Input.Header.Format;	// format
      L     #JobNumber;
      T     "SSA_LOG_Value_Queue".Input.Para_0005;
      L     #processMinute;
      T     "SSA_LOG_Value_Queue".Input.Para_0007;
      L     #StepNumber;
      T     "SSA_LOG_Value_Queue".Input.Para_0008;
      L     #StepTimeMin;
      T     "SSA_LOG_Value_Queue".Input.Para_0009;
// values integer
      L     #EventObject_43;	// event-Nr
      T     "SSA_LOG_Value_Queue".Input.Para_0010;
      L     2;	// object-state going
      T     "SSA_LOG_Value_Queue".Input.Para_0011;
      L     0;	// number additional param
      T     "SSA_LOG_Value_Queue".Input.Para_0012;
// cont log-messages
      L     "SSA_LOG_Value_Queue".Input.Para_0099;	// message counter
      L     1;
      +I;
      T     "SSA_LOG_Value_Queue".Input.Para_0099;	// message counter
// Transform Basic Time to Local Time 
//      CALL  "BT_LT"
//       BT     :="DB Prozesszeit".Arbeitsbereich.dt1
//       WS_DAT :="RegelDB"
//       RET_VAL:=MW218
//       LT     :="RegelDB".LocalTime
// put timestamp into message
      CALL  FC 49 (
           $1                       := 1010,
           $2                       := 18,
           $3                       := 1005,
           $4                       := 462,
           $5                       := 8,
           $6                       := P#M 210.0);
///
      CALL  "SSA_MH_LogEntry_ActValue" (
           DBNumber                 := 1005);
E096: NOP   0;
///     
// Ereignis 44  Kommt         
      A     #EREIGNISBIT_44;
      FP    #Ereignis_44.HP_Kommt;
      JCN   E097;
// header
      L     #MessageType;
      T     "SSA_LOG_Value_Queue".Input.Header.SecType;	// type
      L     #MessageFormat;
      T     "SSA_LOG_Value_Queue".Input.Header.Format;	// format
      L     #JobNumber;
      T     "SSA_LOG_Value_Queue".Input.Para_0005;
      L     #processMinute;
      T     "SSA_LOG_Value_Queue".Input.Para_0007;
      L     #StepNumber;
      T     "SSA_LOG_Value_Queue".Input.Para_0008;
      L     #StepTimeMin;
      T     "SSA_LOG_Value_Queue".Input.Para_0009;
// values integer
      L     #EventObject_44;	// event-Nr
      T     "SSA_LOG_Value_Queue".Input.Para_0010;
      L     1;	// object-state coming
      T     "SSA_LOG_Value_Queue".Input.Para_0011;
      L     0;	// number additional param
      T     "SSA_LOG_Value_Queue".Input.Para_0012;
// cont log-messages
      L     "SSA_LOG_Value_Queue".Input.Para_0099;	// message counter
      L     1;
      +I;
      T     "SSA_LOG_Value_Queue".Input.Para_0099;	// message counter
// Transform Basic Time to Local Time 
//      CALL  "BT_LT"
//       BT     :="DB Prozesszeit".Arbeitsbereich.dt1
//       WS_DAT :="RegelDB"
//       RET_VAL:=MW218
//       LT     :="RegelDB".LocalTime
// put timestamp into message
      CALL  FC 49 (
           $1                       := 1010,
           $2                       := 18,
           $3                       := 1005,
           $4                       := 462,
           $5                       := 8,
           $6                       := P#M 210.0);
///
      CALL  "SSA_MH_LogEntry_ActValue" (
           DBNumber                 := 1005);
E097: NOP   0;
///
// Ereignis 44  Geht        
      A     #EREIGNISBIT_44;
      FN    #Ereignis_44.HP_Geht;
      JCN   E098;
// header
      L     #MessageType;
      T     "SSA_LOG_Value_Queue".Input.Header.SecType;	// type
      L     #MessageFormat;
      T     "SSA_LOG_Value_Queue".Input.Header.Format;	// format
      L     #JobNumber;
      T     "SSA_LOG_Value_Queue".Input.Para_0005;
      L     #processMinute;
      T     "SSA_LOG_Value_Queue".Input.Para_0007;
      L     #StepNumber;
      T     "SSA_LOG_Value_Queue".Input.Para_0008;
      L     #StepTimeMin;
      T     "SSA_LOG_Value_Queue".Input.Para_0009;
// values integer
      L     #EventObject_44;	// event-Nr
      T     "SSA_LOG_Value_Queue".Input.Para_0010;
      L     2;	// object-state going
      T     "SSA_LOG_Value_Queue".Input.Para_0011;
      L     0;	// number additional param
      T     "SSA_LOG_Value_Queue".Input.Para_0012;
// cont log-messages
      L     "SSA_LOG_Value_Queue".Input.Para_0099;	// message counter
      L     1;
      +I;
      T     "SSA_LOG_Value_Queue".Input.Para_0099;	// message counter
// Transform Basic Time to Local Time 
//      CALL  "BT_LT"
//       BT     :="DB Prozesszeit".Arbeitsbereich.dt1
//       WS_DAT :="RegelDB"
//       RET_VAL:=MW218
//       LT     :="RegelDB".LocalTime
// put timestamp into message
      CALL  FC 49 (
           $1                       := 1010,
           $2                       := 18,
           $3                       := 1005,
           $4                       := 462,
           $5                       := 8,
           $6                       := P#M 210.0);
///
      CALL  "SSA_MH_LogEntry_ActValue" (
           DBNumber                 := 1005);
E098: NOP   0;
NETWORK
TITLE =
NETWORK
TITLE = Test-Event
// Ereignis 47 Kommt         
      A     #EREIGNISBIT_47;
      FP    #Ereignis_47.FP_Kommt;
      JCN   E993;
// header
      L     #MessageType;
      T     "SSA_LOG_Value_Queue".Input.Header.SecType;	// type
      L     #MessageFormat;
      T     "SSA_LOG_Value_Queue".Input.Header.Format;	// format
      L     #JobNumber;
      T     "SSA_LOG_Value_Queue".Input.Para_0005;
      L     #processMinute;
      T     "SSA_LOG_Value_Queue".Input.Para_0007;
      L     #StepNumber;
      T     "SSA_LOG_Value_Queue".Input.Para_0008;
      L     #StepTimeMin;
      T     "SSA_LOG_Value_Queue".Input.Para_0009;
// values integer
      L     #EventObject_47;	// event-Nr
      T     "SSA_LOG_Value_Queue".Input.Para_0010;
      L     1;	// object-state coming
      T     "SSA_LOG_Value_Queue".Input.Para_0011;
      L     0;	// number additional param
      T     "SSA_LOG_Value_Queue".Input.Para_0012;
//      CALL  "BT_LT"
//       BT     :="DB Prozesszeit".Arbeitsbereich.dt1
//       WS_DAT :="RegelDB"
//       RET_VAL:=MW218
//       LT     :="RegelDB".LocalTime
      CALL  FC 49 (
           $1                       := 1010,
           $2                       := 18,
           $3                       := 1005,
           $4                       := 462,
           $5                       := 8,
           $6                       := P#M 210.0);
      CALL  "SSA_MH_LogEntry_ActValue" (
           DBNumber                 := 1005);
E993: NOP   0;
// Ereignis 47 Geht
      A     #EREIGNISBIT_47;
      FN    #Ereignis_47.FN_Geht;
      JCN   E994;
// header
      L     #MessageType;
      T     "SSA_LOG_Value_Queue".Input.Header.SecType;	// type
      L     #MessageFormat;
      T     "SSA_LOG_Value_Queue".Input.Header.Format;	// format
      L     #JobNumber;
      T     "SSA_LOG_Value_Queue".Input.Para_0005;
      L     #processMinute;
      T     "SSA_LOG_Value_Queue".Input.Para_0007;
      L     #StepNumber;
      T     "SSA_LOG_Value_Queue".Input.Para_0008;
      L     #StepTimeMin;
      T     "SSA_LOG_Value_Queue".Input.Para_0009;
// values integer
      L     #EventObject_47;	// event-Nr
      T     "SSA_LOG_Value_Queue".Input.Para_0010;
      L     2;	// object-state going
      T     "SSA_LOG_Value_Queue".Input.Para_0011;
      L     0;	// number additional param
      T     "SSA_LOG_Value_Queue".Input.Para_0012;
// cont log-messages
      L     "SSA_LOG_Value_Queue".Input.Para_0099;	// message counter
      L     1;
      +I;
      T     "SSA_LOG_Value_Queue".Input.Para_0099;	// message counter
//      CALL  "BT_LT"
//       BT     :="DB Prozesszeit".Arbeitsbereich.dt1
//       WS_DAT :="RegelDB"
//       RET_VAL:=MW218
//       LT     :="RegelDB".LocalTime
      CALL  FC 49 (
           $1                       := 1010,
           $2                       := 18,
           $3                       := 1005,
           $4                       := 462,
           $5                       := 8,
           $6                       := P#M 210.0);
      CALL  "SSA_MH_LogEntry_ActValue" (
           DBNumber                 := 1005);
E994: NOP   0;
NETWORK
TITLE =
//Blinker zum testen
      AN    T 29;
      L     S5T#2S;
      SD    T 28;
      A     T 28;
      L     S5T#2S;
      SD    T 29;
      CLR;
      =     M 300.0;
NETWORK
TITLE =
      BE;
END_FUNCTION_BLOCK

FUNCTION_BLOCK "SSA_FU_Siemens"	// FB 1811
TITLE = Siemens FU/SEW
//COPYRIGHT:    (C) 2004  BUHLER AG, CH-9240 UZWIL, SWITZERLAND
//
//PRODUCT:      SSA
//
//TITLE:        Communication  Siemens FU SEW_MOVIDRIVE
//
//--------------------------------------------------------------------------------
//
//IDENT:         AUTHOR:             DEPT:                            DATE:
//
//FB1902.1.0     A.Egli              CT3                              13-Jul-2007
//               1st Release
//
//--------------------------------------------------------------------------------
//
//PURPOSE: 
//
//MANUAL : 
//
//RESTRICTIONS: 
//
//--------------------------------------------------------------------------------
//
AUTHOR : PE
FAMILY : STD
VERSION : 0.0
VAR
  spare1 : INT ;
  InEnableRev : BOOL ;
  InEnableFwd : BOOL ;
  CmdFaultReset : BOOL ;
  OutRunningRev : BOOL ;	//Feedback for element motor
  OutRunningFwd : BOOL ;	//Feedback for element motor
  OutFault : BOOL ;	//Feedback for element motor
  spare2 : INT ;
  Input : STRUCT
   StateWord_1 : STRUCT 	//Statuswort MOVIDRIVE
    STATE_WORD_BIT_8 : BOOL ;
    STATE_WORD_BIT_9 : BOOL ;
    STATE_WORD_BIT_10 : BOOL ;
    STATE_WORD_BIT_11 : BOOL ;
    STATE_WORD_BIT_12 : BOOL ;
    STATE_WORD_BIT_13 : BOOL ;
    STATE_WORD_BIT_14 : BOOL ;
    STATE_WORD_BIT_15 : BOOL ;
    ENDSTUFE_FREIGEGEBEN : BOOL ;
    BETRIEBSBEREIT : BOOL ;
    PA_DATEN_FREIGEGEBEN : BOOL ;
    AKTUELL_INTEGRATORSATZ : BOOL ;
    AKTUELL_PARAMETERSATZ : BOOL ;
    STOERUNG_WARNUNG : BOOL ;
    LS_RECHTS_AKTIV : BOOL ;
    LS_LINKS_AKTIV : BOOL ;
   END_STRUCT ;
   ActualValue01 : INT ;	//Hauptistwert / Prozessdaten PD2
   ActualValue02 : INT ;	//Prozessdaten PD3
   ActualValue03 : INT ;	//Prozessdaten PD4
   ActualValue04 : INT ;	//Prozessdaten PD5
   ActualValue05 : INT ;	//Prozessdaten PD6
  END_STRUCT ;
  Output : STRUCT
   ControlWord_1 : STRUCT 	//Steuerwort MOVIDRIVE
    CONTROL_WORD_BIT_8 : BOOL ;
    CONTROL_WORD_BIT_9 : BOOL ;
    CONTROL_WORD_BIT_10 : BOOL ;
    CONTROL_WORD_BIT_11 : BOOL ;
    CONTROL_WORD_BIT_12 : BOOL ;
    CONTROL_WORD_BIT_13 : BOOL ;
    CONTROL_WORD_BIT_14 : BOOL ;
    CONTROL_WORD_BIT_15 : BOOL ;
    CONTROL_WORD_BIT_0 : BOOL ;
    CONTROL_WORD_BIT_1 : BOOL ;
    CONTROL_WORD_BIT_2 : BOOL ;
    CONTROL_WORD_BIT_3 : BOOL ;
    CONTROL_WORD_BIT_4 : BOOL ;
    CONTROL_WORD_BIT_5 : BOOL ;
    CONTROL_WORD_BIT_6 : BOOL ;
    CONTROL_WORD_BIT_7 : BOOL ;
   END_STRUCT ;
   SetpointValue01 : INT ;	//Hauptsollwert / Prozessdaten PD2
   SetpointValue02 : INT ;	//Prozessdaten PD3
   SetpointValue03 : INT ;	//Prozessdaten PD4
   SetpointValue04 : INT ;	//Prozessdaten PD5
   SetpointValue05 : INT ;	//Prozessdaten PD6
  END_STRUCT ;
  Par : STRUCT
   spare1 : INT ;
   spare2 : INT ;
   spare3 : INT ;
   ParMovidrive : BOOL ;
   ParSinamics : BOOL ;
   ParMicromaster : BOOL ;
   ParABB : BOOL ;
   ParNord : BOOL ;
   Danfoss : BOOL ;
   ParIOByteNo : INT ;
  END_STRUCT ;
END_VAR
VAR_TEMP
  tmpAddrDB : INT ;
  tmpAddrIO : DINT ;
  tmpAddrInputFU : DINT ;
  tmpAddrOutputFU : DINT ;
  MM_StateWord : STRUCT 	//Statuswort Micromaster
   DREHZAHL_ABWEICHUNG_OK : BOOL ;	//0=Nicht im Toleranzband             1=Soll-Ist-Überwachung im Toleranzband
   FUEHRUNG : BOOL ;	//0=Fuehrung Lokal                    1=Fuehrung SPS
   VERGLEICHSWERT : BOOL ;	//0=Vergleichswert nicht erreicht     1=Vergleichswert erreicht/ueberschritten
   GRENZE_ERREICHT : BOOL ;	//0=I-, M- oder P-Grenze erreicht     1=I-, M- oder P-Grenze nicht erreicht
   HALTEBREMSE : BOOL ;	//0=Motor Haltebremse                 1=Steuern Haltebremse
   WARN_UEBERTEMP_MOTOR : BOOL ;	//0=Warnung nicht wirksam             1=Warnung Übertemperatur Motor wirksam
   DREH_RECHTS : BOOL ;	//0=Linkslauf                         1=Rechtslauf
   WARNUNG_UEBERTEMP_FU : BOOL ;	//0=Warnung thermische Überlast Umrichter 1=Keine Warnung wirksam
   EINSCHALTBEREIT : BOOL ;	//0=Nicht einschaltbereit             1=Einschaltbereit
   BETRIEBSBEREIT : BOOL ;	//0=Nicht betriebsbereit              1=Betriebsbereit
   BETRIEB_FREIGEGEBEN : BOOL ;	//0=Betrieb gesperrt   1=Betrieb freigegeben->Hochlauf auf anliegendem Sollwert
   STOERUNG : BOOL ;	//0=Keine Störung wirksam             1=Störung wirksam
   AUS_2 : BOOL ;	//0=Austrudeln aktiv (AUS2)           1=Kein AUS2 aktiv
   AUS_3 : BOOL ;	//0=Schnellhalt aktiv (AUS3)          1=Kein AUS3 aktiv
   EINSCHALTSPERRE : BOOL ;	//1=Einschaltsperre -> Wiedereinschalten durch AUS1 und anschließendes EIN
   WARNUNG : BOOL ;	//0=Keine Warnung wirksam             1=Warnung wirksam, Motor weiter im Betrieb
  END_STRUCT ;
  MM_ControlWord : STRUCT 	//Steuerwort Micromaster
   TIPPEN_RECHTS : BOOL ;	//1=Tippen rechts
   TIPPEN_LINKS : BOOL ;	//1=Tippen links
   PZD_GUELTIG : BOOL ;	//0=Sollwerte ungueltig              1=Sollwerte gueltig
   DREHRICHTUNGSUMKEHR : BOOL ;	//Drehrichtungsumkehr: 0=Rechtsdrehfeld / 1=Linksdrehfeld
   CONTROL_WORD_BIT_12 : BOOL ;	//reserviert
   MOTOR_POTI_HIGH : BOOL ;	//1=Motorpotentiometer höher
   MOTOR_POTI_DOWN : BOOL ;	//1=Motorpotentiometer tiefer
   LOCAL : BOOL ;	//0=Fern-Steuerung aktiv             1=Vorort-Steuerung aktiv
   AUS1 : BOOL ;	//0=AUS1->Abbremsen an der Rücklauframpe   1=EIN
   AUS2 : BOOL ;	//0=Austrudeln (AUS2)                      1=kein Austrudeln
   AUS3 : BOOL ;	//0=Schnellhalt (AUS3)->Abbremsen an der Schnellhalt-Rampe  1=kein Schnellhalt
   BETRIEB_FREIGEBEN : BOOL ;	//0=Betrieb sperren        1=Betrieb freigeben->Hochlauf mit anliegendem Sollwert
   HOCHLAUF_SPERREN : BOOL ;	//0=Hochlaufgeber wird auf NULL gesetzt    1=Hochlaufgeber freigeben
   HOCHLAUF_STOPPEN : BOOL ;	//0=Hochlaufgeber einfrieren               1=Hochlaufgeber freigeben
   SOLLWERT_FREIGEBEN : BOOL ;	//0=Drehzahlsollwert wird auf NULL gesetzt 1=Drehzahlsollwert freigeben
   FEHLER_QUITTIEREN : BOOL ;	//Flanke 0 -> 1 = Fehler quittieren, quittiert alle aktuellen Störungen
  END_STRUCT ;
  MD_StateWord : STRUCT 	//Statuswort MOVIDRIVE
   STATE_WORD_BIT_8 : BOOL ;	//Geraetezustand / Fehelr-Nummer
   STATE_WORD_BIT_9 : BOOL ;	//Geraetezustand / Fehelr-Nummer
   STATE_WORD_BIT_10 : BOOL ;	//Geraetezustand / Fehelr-Nummer
   STATE_WORD_BIT_11 : BOOL ;	//Geraetezustand / Fehelr-Nummer
   STATE_WORD_BIT_12 : BOOL ;	//Geraetezustand / Fehelr-Nummer
   STATE_WORD_BIT_13 : BOOL ;	//Geraetezustand / Fehelr-Nummer
   STATE_WORD_BIT_14 : BOOL ;	//Geraetezustand / Fehelr-Nummer
   STATE_WORD_BIT_15 : BOOL ;	//Geraetezustand / Fehelr-Nummer
   ENDSTUFE_FREIGEGEBEN : BOOL ;	//0=Endstufe gesperrt                 1=Endstufe freigegeben
   BETRIEBSBEREIT : BOOL ;	//0=Umrichter nicht betriebsbereit    1=Umrichter betriebsbereit
   PA_DATEN_FREIGEGEBEN : BOOL ;	//0=PA-Daten gesperrt                 1=PA-Daten freigegeben
   AKTUELL_INTEGRATORSATZ : BOOL ;	//0=Integrator 1                      1=Integrator 2
   AKTUELL_PARAMETERSATZ : BOOL ;	//0=Parametersatz 1                   1=Parametersatz 2
   STOERUNG_WARNUNG : BOOL ;	//0=keine Störung/Warnung             1=Störung/Warnung
   LS_RECHTS_AKTIV : BOOL ;	//1=Endschalter RECHTS betaetigt -> Drehrichtung RECHTS gesperrt
   LS_LINKS_AKTIV : BOOL ;	//1=Endschalter LINKS betaetigt -> Drehrichtung LINKS gesperrt
  END_STRUCT ;
  MD_ControlWord : STRUCT 	//Steuerwort MOVIDRIVE
   CONTROL_WORD_BIT_8 : BOOL ;	//Reserviert für Zusatzfuktionen = "0"
   CONTROL_WORD_BIT_9 : BOOL ;	//Reserviert für Zusatzfuktionen = "0"
   CONTROL_WORD_BIT_10 : BOOL ;	//Reserviert für Zusatzfuktionen = "0"
   CONTROL_WORD_BIT_11 : BOOL ;	//Reserviert für Zusatzfuktionen = "0"
   CONTROL_WORD_BIT_12 : BOOL ;	//Reserviert für Zusatzfuktionen = "0"
   CONTROL_WORD_BIT_13 : BOOL ;	//Reserviert für Zusatzfuktionen = "0"
   CONTROL_WORD_BIT_14 : BOOL ;	//Reserviert für Zusatzfuktionen = "0"
   CONTROL_WORD_BIT_15 : BOOL ;	//Reserviert für Zusatzfuktionen = "0"
   REGLERSPERRE : BOOL ;	//0=Freigabe                          1=Regler sperren, Bremse aktivieren
   FREIGABE_SCHNELLSTOPP : BOOL ;	//0=Schnellstopp                      1=Freigabe
   FREIGABE_HALT : BOOL ;	//0=Halt an Integrator/Prozess-Rampe  1=Freigabe
   HALTEREGELUNG : BOOL ;	//0=Halteregelung nicht aktiv         1=Halteregelung aktiv
   INTEGRATOR : BOOL ;	//0=Integrator 1                      1=Integrator 2
   PARAMETERSATZ : BOOL ;	//0=Parametersatz 1                   1=Parametersatz 2
   RESET : BOOL ;	//0=nicht aktiv                       1=Fehler quittieren
   RESERVE_BIT_7 : BOOL ;	//Reserviert für Zusatzfuktionen = "0"
  END_STRUCT ;
  SI_StateWord : STRUCT 	//Statuswort Sinamics
   DREHZAHL_ABWEICHUNG_OK : BOOL ;	//0=Nicht im Toleranzband             1=Soll-Ist-Überwachung im Toleranzband
   FUEHRUNG : BOOL ;	//0=Fuehrung Lokal                    1=Fuehrung SPS
   VERGLEICHSWERT : BOOL ;	//0=Vergleichswert nicht erreicht     1=Vergleichswert erreicht/ueberschritten
   GRENZE_ERREICHT : BOOL ;	//0=I-, M- oder P-Grenze erreicht     1=I-, M- oder P-Grenze nicht erreicht
   STATE_WORD_BIT_12 : BOOL ;	//reserviert
   WARN_UEBERTEMP_MOTOR : BOOL ;	//0=Warnung nicht wirksam             1=Warnung Übertemperatur Motor wirksam
   DREH_RECHTS : BOOL ;	//0=Motor dreht nicht vorwärts        1=Motor dreht vorwärts
   WARNUNG_UEBERTEMP_FU : BOOL ;	//0=Warnung thermische Überlast Umrichter 1=Keine Warnung wirksam
   EINSCHALTBEREIT : BOOL ;	//0=Nicht einschaltbereit             1=Einschaltbereit
   BETRIEBSBEREIT : BOOL ;	//0=Nicht betriebsbereit              1=Betriebsbereit
   BETRIEB_FREIGEGEBEN : BOOL ;	//0=Betrieb gesperrt   1=Betrieb freigegeben->Hochlauf auf anliegendem Sollwert
   STOERUNG : BOOL ;	//0=Keine Störung wirksam             1=Störung wirksam
   AUS_2 : BOOL ;	//0=Austrudeln aktiv (AUS2)           1=Kein AUS2 aktiv
   AUS_3 : BOOL ;	//0=Schnellhalt aktiv (AUS3)          1=Kein AUS3 aktiv
   EINSCHALTSPERRE : BOOL ;	//1=Einschaltsperre -> Wiedereinschalten durch AUS1 und anschließendes EIN
   WARNUNG : BOOL ;	//0=Keine Warnung wirksam             1=Warnung wirksam
  END_STRUCT ;
  SI_ControlWord : STRUCT 	//Statuswort Sinamics
   CONTROL_WORD_BIT_8 : BOOL ;	//reserviert
   CONTROL_WORD_BIT_9 : BOOL ;	//reserviert
   PZD_GUELTIG : BOOL ;	//Steuerworte, Sollwerte vom Profibus werden: 0=nicht ausgewertet / 1=ausgewertet
   DREHRICHTUNGSUMKEHR : BOOL ;	//Drehrichtungsumkehr: 0=Rechtsdrehfeld / 1=Linksdrehfeld
   CONTROL_WORD_BIT_12 : BOOL ;	//reserviert
   MOTOR_POTI_HIGH : BOOL ;	//1=Motorpotentiometer höher
   MOTOR_POTI_DOWN : BOOL ;	//1=Motorpotentiometer tiefer
   CONTROL_WORD_BIT_15 : BOOL ;	//reserviert
   AUS1 : BOOL ;	//0=AUS1->Abbremsen an der Rücklauframpe   1=EIN
   AUS2 : BOOL ;	//0=Austrudeln (AUS2)                      1=kein Austrudeln
   AUS3 : BOOL ;	//0=Schnellhalt (AUS3)->Abbremsen an der Schnellhalt-Rampe  1=kein Schnellhalt
   BETRIEB_FREIGEBEN : BOOL ;	//0=Betrieb sperren        1=Betrieb freigeben->Hochlauf mit anliegendem Sollwert
   HOCHLAUF_SPERREN : BOOL ;	//0=Hochlaufgeber wird auf NULL gesetzt    1=Hochlaufgeber freigeben
   HOCHLAUF_STOPPEN : BOOL ;	//0=Hochlaufgeber einfrieren               1=Hochlaufgeber wiederaufsetzen
   SOLLWERT_FREIGEBEN : BOOL ;	//0=Drehzahlsollwert wird auf NULL gesetzt 1=Drehzahlsollwert freigeben
   FEHLER_QUITTIEREN : BOOL ;	//Flanke 0 -> 1 = Fehler quittieren, quittiert alle aktuellen Störungen
  END_STRUCT ;
END_VAR
BEGIN
NETWORK
TITLE = Calculate Address of Inverter
      L     #Par.ParIOByteNo;
      SLD   3;
      T     #tmpAddrIO;
      L     P##Input;
      L     DW#16#FFFFFF;
      AD;
      TAR2;
      +D;
      T     #tmpAddrInputFU;
      L     P##Output;
      L     DW#16#FFFFFF;
      AD;
      TAR2;
      +D;
      T     #tmpAddrOutputFU;
NETWORK
TITLE = Prepare Commands Par.ParMovidrive
      AN    #Par.ParMovidrive;
      JC    MDJ0;
//Load Status Word
      LAR1  #tmpAddrInputFU;
      L     DIW [AR1,P#0.0];	//Status Word
      LAR1  P##MD_StateWord;
      T     LW [AR1,P#0.0];	// MD_StateWord
// prepare steuerword
      L     W#16#2;	// FREIGABE_SCHNELLSTOPP=1; FREIGABE_HALT=0
      A     #InEnableFwd;
      JCN   MDJ1;
      L     W#16#6;	// FREIGABE_SCHNELLSTOPP=1; FREIGABE_HALT=1
MDJ1: LAR1  #tmpAddrOutputFU;
      T     DIW [AR1,P#0.0];	// controlword 
//-----------------------------------------
// Fault Reset ins Steuerwort
      A     #CmdFaultReset;
      A     #Input.StateWord_1.STOERUNG_WARNUNG;	// Fehler von FU
      JCN   MDR1;
      L     W#16#40;	// RESET=1; FREIGABE_SCHNELLSTOPP=0; FREIGABE_HALT=0
      LAR1  #tmpAddrOutputFU;
      T     DIW [AR1,P#0.0];	// controlword 
MDR1: NOP   0;
//- Feedback for motor
      A     #MD_StateWord.BETRIEBSBEREIT;
      A     #MD_StateWord.PA_DATEN_FREIGEGEBEN;
      AN    #MD_StateWord.STOERUNG_WARNUNG;
      =     #OutRunningRev;
      A     #MD_StateWord.BETRIEBSBEREIT;
      A     #MD_StateWord.PA_DATEN_FREIGEGEBEN;
      AN    #MD_StateWord.STOERUNG_WARNUNG;
      =     #OutRunningFwd;
      A     #MD_StateWord.STOERUNG_WARNUNG;
      =     #OutFault;
MDJ0: NOP   0;
NETWORK
TITLE = Prepare Commands Par.ParMicroMaster
      AN    #Par.ParNord;
      JC    MMJ0;
//Load Status Word
      LAR1  #tmpAddrInputFU;
      L     DIW [AR1,P#0.0];	//Status Word
      LAR1  P##MM_StateWord;
      T     LW [AR1,P#0.0];	// MM_StateWord
// prepare steuerword
      L     W#16#47E;	// Stop=AUS1
      A     #InEnableFwd;
      JCN   MMJ1;
      L     W#16#47F;	// Start=EIN
MMJ1: LAR1  #tmpAddrOutputFU;
      T     DIW [AR1,P#0.0];	// controlword 
//-----------------------------------------
// Fault Reset ins Steuerwort
      A     #CmdFaultReset;
      A     #Input.StateWord_1.STOERUNG_WARNUNG;	// Fehler von FU
      JCN   MMR1;
      L     W#16#4FE;	// Reset ins Steuerwort
      LAR1  #tmpAddrOutputFU;
      T     DIW [AR1,P#0.0];	// controlword 
MMR1: NOP   0;
//- Feedback for motor
      A     #MM_StateWord.BETRIEBSBEREIT;
      AN    #MM_StateWord.STOERUNG;
      A     #InEnableRev;
      =     #OutRunningRev;
      A     #MM_StateWord.BETRIEBSBEREIT;
      AN    #MM_StateWord.STOERUNG;
      A     #InEnableFwd;
      =     #OutRunningFwd;
      A     #MM_StateWord.STOERUNG;
      =     #OutFault;
MMJ0: NOP   0;
NETWORK
TITLE = Prepare Commands Par.ParSinamics
      AN    #Par.ParSinamics;
      JC    SIJ0;
//Load Status Word
      LAR1  #tmpAddrInputFU;
      L     DIW [AR1,P#0.0];	//Status Word
      LAR1  P##MM_StateWord;
      T     LW [AR1,P#0.0];	// MM_StateWord
// prepare steuerword
      L     W#16#47E;	// Stop=AUS1
      A     #InEnableFwd;
      JCN   SIJ1;
      L     W#16#47F;	// Start=EIN
SIJ1: LAR1  #tmpAddrOutputFU;
      T     DIW [AR1,P#0.0];	// controlword 
//-----------------------------------------
// Fault Reset ins Steuerwort
      A     #CmdFaultReset;
      A     #Input.StateWord_1.STOERUNG_WARNUNG;	// Fehler von FU
      JCN   SIR1;
      L     W#16#4FE;	// Reset ins Steuerwort
      LAR1  #tmpAddrOutputFU;
      T     DIW [AR1,P#0.0];	// controlword 
SIR1: NOP   0;
//- Feedback for motor
      A     #SI_StateWord.BETRIEBSBEREIT;
      AN    #SI_StateWord.STOERUNG;
      A     #InEnableRev;
      =     #OutRunningRev;
      A     #SI_StateWord.BETRIEBSBEREIT;
      AN    #SI_StateWord.STOERUNG;
      A     #InEnableFwd;
      =     #OutRunningFwd;
      A     #SI_StateWord.STOERUNG;
      =     #OutFault;
SIJ0: NOP   0;
NETWORK
TITLE =
      A     #CmdFaultReset;
      R     #CmdFaultReset;
NETWORK
TITLE = Read Inputs of Inverter
      LAR1  #tmpAddrIO;
      L     PID [AR1,P#0.0];
      LAR1  #tmpAddrInputFU;
      T     DID [AR1,P#0.0];
      LAR1  #tmpAddrIO;
      L     PID [AR1,P#4.0];
      LAR1  #tmpAddrInputFU;
      T     DID [AR1,P#4.0];
      LAR1  #tmpAddrIO;
      L     PID [AR1,P#8.0];
      LAR1  #tmpAddrInputFU;
      T     DID [AR1,P#8.0];
NETWORK
TITLE = Write Outputs of Inverter
      LAR1  #tmpAddrOutputFU;
      L     DID [AR1,P#0.0];
      LAR1  #tmpAddrIO;
      T     PQD [AR1,P#0.0];
      LAR1  #tmpAddrOutputFU;
      L     DID [AR1,P#4.0];
      LAR1  #tmpAddrIO;
      T     PQD [AR1,P#4.0];
      LAR1  #tmpAddrOutputFU;
      L     DID [AR1,P#8.0];
      LAR1  #tmpAddrIO;
      T     PQD [AR1,P#8.0];
NETWORK
TITLE =
      BE;
END_FUNCTION_BLOCK

FUNCTION_BLOCK "SSA_SEW_MOVIDRIVE"	// FB 1812
TITLE = SEW MOVIDRIVE
//COPYRIGHT:    (C) 2004  BUHLER AG, CH-9240 UZWIL, SWITZERLAND
//
//PRODUCT:      SSA
//
//TITLE:        SEW MOVIDRIVE Frequency Inverter Profibus Communication
//
//--------------------------------------------------------------------------------
//
//IDENT:         AUTHOR:             DEPT:                            DATE:
//
//FB1812.2.0     M.Wedler            AEB41                            25-Okt-2007
//               2nd Release
//FB1811.1.0     A.Egli              CT3                              13-Jul-2007
//               1st Release
//
//--------------------------------------------------------------------------------
//
//PURPOSE: 
//
//MANUAL : 
//
//RESTRICTIONS: 
//
//--------------------------------------------------------------------------------
//
AUTHOR : MW
FAMILY : STD
VERSION : 0.0
VAR
  InValuePC : INT ;	//Aktuel value 1 in [0.01 %]
  InEnableRev : BOOL ;
  InEnableFwd : BOOL ;
  CmdFaultReset : BOOL ;
  OutRunningRev : BOOL ;	//Feedback for element motor
  OutRunningFwd : BOOL ;	//Feedback for element motor
  OutFault : BOOL ;	//Feedback for element motor
  MotorStStopped : BOOL ;	//Motor has come to a standstill after stopping time
  Spare : BOOL ;
  OutValuePC : INT ;	//Setpoint value 1 in [0.01 %]
  Input : STRUCT
   StateWord_1 : STRUCT 	//Statuswort MOVIDRIVE
    STATE_WORD_BIT_8 : BOOL ;	//Geraetezustand / Fehelr-Nummer
    STATE_WORD_BIT_9 : BOOL ;	//Geraetezustand / Fehelr-Nummer
    STATE_WORD_BIT_10 : BOOL ;	//Geraetezustand / Fehelr-Nummer
    STATE_WORD_BIT_11 : BOOL ;	//Geraetezustand / Fehelr-Nummer
    STATE_WORD_BIT_12 : BOOL ;	//Geraetezustand / Fehelr-Nummer
    STATE_WORD_BIT_13 : BOOL ;	//Geraetezustand / Fehelr-Nummer
    STATE_WORD_BIT_14 : BOOL ;	//Geraetezustand / Fehelr-Nummer
    STATE_WORD_BIT_15 : BOOL ;	//Geraetezustand / Fehelr-Nummer
    ENDSTUFE_FREIGEGEBEN : BOOL ;	//0=Endstufe gesperrt                 1=Endstufe freigegeben
    BETRIEBSBEREIT : BOOL ;	//0=Umrichter nicht betriebsbereit    1=Umrichter betriebsbereit
    PA_DATEN_FREIGEGEBEN : BOOL ;	//0=PA-Daten gesperrt                 1=PA-Daten freigegeben
    AKTUELL_INTEGRATORSATZ : BOOL ;	//0=Integrator 1                      1=Integrator 2
    AKTUELL_PARAMETERSATZ : BOOL ;	//0=Parametersatz 1                   1=Parametersatz 2
    STOERUNG_WARNUNG : BOOL ;	//0=keine Störung/Warnung             1=Störung/Warnung
    LS_RECHTS_AKTIV : BOOL ;	//1=Endschalter RECHTS betaetigt -> Drehrichtung RECHTS gesperrt
    LS_LINKS_AKTIV : BOOL ;	//1=Endschalter LINKS betaetigt -> Drehrichtung LINKS gesperrt
   END_STRUCT ;
   ActualValue01 : INT ;	//Hauptistwert / Prozessdaten PD2
   ActualValue02 : INT ;	//Prozessdaten PD3
   ActualValue03 : INT ;	//Prozessdaten PD4
   ActualValue04 : INT ;	//Prozessdaten PD5
   ActualValue05 : INT ;	//Prozessdaten PD6
  END_STRUCT ;
  Output : STRUCT
   ControlWord_1 : STRUCT 	//Steuerwort MOVIDRIVE
    CONTROL_WORD_BIT_8 : BOOL ;	//Reserviert für Zusatzfuktionen = "0"
    CONTROL_WORD_BIT_9 : BOOL ;	//Reserviert für Zusatzfuktionen = "0"
    CONTROL_WORD_BIT_10 : BOOL ;	//Reserviert für Zusatzfuktionen = "0"
    CONTROL_WORD_BIT_11 : BOOL ;	//Reserviert für Zusatzfuktionen = "0"
    CONTROL_WORD_BIT_12 : BOOL ;	//Reserviert für Zusatzfuktionen = "0"
    CONTROL_WORD_BIT_13 : BOOL ;	//Reserviert für Zusatzfuktionen = "0"
    CONTROL_WORD_BIT_14 : BOOL ;	//Reserviert für Zusatzfuktionen = "0"
    CONTROL_WORD_BIT_15 : BOOL ;	//Reserviert für Zusatzfuktionen = "0"
    REGLERSPERRE : BOOL ;	//0=Freigabe                          1=Regler sperren, Bremse aktivieren
    FREIGABE_SCHNELLSTOPP : BOOL ;	//0=Schnellstopp                      1=Freigabe
    FREIGABE_HALT : BOOL ;	//0=Halt an Integrator/Prozess-Rampe  1=Freigabe
    HALTEREGELUNG : BOOL ;	//0=Halteregelung nicht aktiv         1=Halteregelung aktiv
    INTEGRATOR : BOOL ;	//0=Integrator 1                      1=Integrator 2
    PARAMETERSATZ : BOOL ;	//0=Parametersatz 1                   1=Parametersatz 2
    RESET : BOOL ;	//0=nicht aktiv                       1=Fehler quittieren
    RESERVE_BIT_7 : BOOL ;	//Reserviert für Zusatzfuktionen = "0"
   END_STRUCT ;
   SetpointValue01 : INT ;	//Hauptsollwert / Prozessdaten PD2
   SetpointValue02 : INT ;	//Prozessdaten PD3
   SetpointValue03 : INT ;	//Prozessdaten PD4
   SetpointValue04 : INT ;	//Prozessdaten PD5
   SetpointValue05 : INT ;	//Prozessdaten PD6
  END_STRUCT ;
  Par : STRUCT
   spare1 : INT ;
   spare2 : INT ;
   spare3 : INT ;
   ParMovidrive : BOOL ;
   ParSinamics : BOOL ;
   ParMicromaster : BOOL ;
   ParABB : BOOL ;
   ParNord : BOOL ;
   ParDanfoss : BOOL ;
   ParIOByteNo : INT ;
  END_STRUCT ;
END_VAR
VAR_TEMP
  tmpAddrDB : INT ;
  tmpAddrIO : DINT ;
  tmpAddrInputFU : DINT ;
  tmpAddrOutputFU : DINT ;
END_VAR
BEGIN
NETWORK
TITLE = Calculate Address of Inverter
      L     #Par.ParIOByteNo;
      SLD   3;
      T     #tmpAddrIO;
      L     P##Input;
      L     DW#16#FFFFFF;
      AD;
      TAR2;
      +D;
      T     #tmpAddrInputFU;
      L     P##Output;
      L     DW#16#FFFFFF;
      AD;
      TAR2;
      +D;
      T     #tmpAddrOutputFU;
NETWORK
TITLE = Prepare Commands Par.ParMovidrive
      AN    #Par.ParMovidrive;
      JC    MDJ0;
//Load Status Word
//      LAR1  #tmpAddrInputFU
//      L     DIW [AR1,P#0.0]             //Status Word
//      LAR1  P##MD_StateWord
//      T     LW [AR1,P#0.0]              // MD_StateWord
// prepare steuerword
      L     W#16#2;	// FREIGABE_SCHNELLSTOPP=1; FREIGABE_HALT=0
      A     #InEnableFwd;
      O     #InEnableRev;
      JCN   MDJ1;
      L     W#16#6;	// FREIGABE_SCHNELLSTOPP=1; FREIGABE_HALT=1
MDJ1: LAR1  #tmpAddrOutputFU;
      T     DIW [AR1,P#0.0];	// controlword 
//-----------------------------------------
// Fault Reset ins Steuerwort
      A     #CmdFaultReset;
      A     #Input.StateWord_1.STOERUNG_WARNUNG;	// Fehler von FU
      JCN   MDR1;
      L     W#16#40;	// RESET=1; FREIGABE_SCHNELLSTOPP=0; FREIGABE_HALT=0
      LAR1  #tmpAddrOutputFU;
      T     DIW [AR1,P#0.0];	// controlword 
MDR1: NOP   0;
//- Feedback for motor
      A     #Input.StateWord_1.BETRIEBSBEREIT;
      A     #Input.StateWord_1.PA_DATEN_FREIGEGEBEN;
      AN    #Input.StateWord_1.STOERUNG_WARNUNG;
      =     #OutRunningRev;
      A     #Input.StateWord_1.BETRIEBSBEREIT;
      A     #Input.StateWord_1.PA_DATEN_FREIGEGEBEN;
      AN    #Input.StateWord_1.STOERUNG_WARNUNG;
      =     #OutRunningFwd;
      A     #Input.StateWord_1.STOERUNG_WARNUNG;
      =     #OutFault;
NETWORK
TITLE = Prepare setpoint value
//Motor nominal speed:
//C000H = -16384Dez = -100.0% (direction left)
//4000H = +16384Dez = +100.0% (direction right)
      L     #OutValuePC;
      ITD;
      DTR;
      L     1.638400e+00;
      *R;
      RND;
      A     #InEnableRev;
      JCN   tsp;
      NEGD;
tsp:  T     #Output.SetpointValue01;
NETWORK
TITLE = Prepare actual value
//Motor nominal speed:
//C000H = -16384Dez = -100.0% (direction left)
//4000H = +16384Dez = +100.0% (direction right)
      L     #Input.ActualValue01;
      ITD;
      DTR;
      ABS;
      L     1.638400e+00;
      /R;
      RND;
      T     #InValuePC;
NETWORK
TITLE =
      A     #CmdFaultReset;
      R     #CmdFaultReset;
NETWORK
TITLE = Read Inputs of Inverter
//      LAR1  #tmpAddrIO
//      L     PED [AR1,P#0.0]
//      LAR1  #tmpAddrInputFU
//      T     DID [AR1,P#0.0]
//      LAR1  #tmpAddrIO
//      L     PED [AR1,P#4.0]
//      LAR1  #tmpAddrInputFU
//      T     DID [AR1,P#4.0]
//      LAR1  #tmpAddrIO
//      L     PED [AR1,P#8.0]
//      LAR1  #tmpAddrInputFU
//      T     DID [AR1,P#8.0]
// 3 Process Data Words  // [2.0]
      LAR1  #tmpAddrIO;
      L     PIW [AR1,P#0.0];
      LAR1  #tmpAddrInputFU;
      T     DIW [AR1,P#0.0];
      LAR1  #tmpAddrIO;
      L     PIW [AR1,P#2.0];
      LAR1  #tmpAddrInputFU;
      T     DIW [AR1,P#2.0];
      LAR1  #tmpAddrIO;
      L     PIW [AR1,P#4.0];
      LAR1  #tmpAddrInputFU;
      T     DIW [AR1,P#4.0];
NETWORK
TITLE = Write Outputs of Inverter
//      LAR1  #tmpAddrOutputFU
//      L     DID [AR1,P#0.0]
//      LAR1  #tmpAddrIO
//      T     PAD [AR1,P#0.0]
//      LAR1  #tmpAddrOutputFU
//      L     DID [AR1,P#4.0]
//      LAR1  #tmpAddrIO
//      T     PAD [AR1,P#4.0]
//      LAR1  #tmpAddrOutputFU
//      L     DID [AR1,P#8.0]
//      LAR1  #tmpAddrIO
//      T     PAD [AR1,P#8.0]
// 3 Process Data Words  // [2.0]
      LAR1  #tmpAddrOutputFU;
      L     DIW [AR1,P#0.0];
      LAR1  #tmpAddrIO;
      T     PQW [AR1,P#0.0];
      LAR1  #tmpAddrOutputFU;
      L     DIW [AR1,P#2.0];
      LAR1  #tmpAddrIO;
      T     PQW [AR1,P#2.0];
      LAR1  #tmpAddrOutputFU;
      L     DIW [AR1,P#4.0];
      LAR1  #tmpAddrIO;
      T     PQW [AR1,P#4.0];
NETWORK
TITLE =
MDJ0: NOP   0;
      BE;
END_FUNCTION_BLOCK

